	17118:
		F_ADSErrorCodeExt := 'Coupling conditions of synchronization generator incorrect';

	17119:
		F_ADSErrorCodeExt := 'Moving profile of synchronization generator declines dynamic limit of slave axis or required characteristic of profile';

	17120:
		F_ADSErrorCodeExt := 'The encoder generator parameter is not allowed.';

	17121:
		F_ADSErrorCodeExt := 'The external (Fifo) generator parameter is not allowed.';

	17122:
		F_ADSErrorCodeExt := 'The external generator cannot be started, as it is already active.';

	17123:
		F_ADSErrorCodeExt := 'The external generator cannot be stopped, as it is not active.';

	17124:
		F_ADSErrorCodeExt := 'NC-Block with auxiliary axis violates software limit switches of the group.';

	17125:
		F_ADSErrorCodeExt := 'NC-Block type Bezier spline curve contains a cusp (singularity). The Bezier spline curve contain a cusp.';

	17127:
		F_ADSErrorCodeExt := 'Value FOR dead TIME compensation NOT allowed.';

	17128:
		F_ADSErrorCodeExt := 'GROUPERR_RANGE_NOMOTIONWINDOW';

	17129:
		F_ADSErrorCodeExt := 'GROUPERR_RANGE_NOMOTIONFILTERTIME';

	17130:
		F_ADSErrorCodeExt := 'GROUPERR_RANGE_TIMEUNITFIFO';

	17131:
		F_ADSErrorCodeExt := 'GROUPERR_RANGE_OVERRIDETYPE';

	17132:
		F_ADSErrorCodeExt := 'GROUPERR_RANGE_OVERRIDECHANGETIME';

	17133:
		F_ADSErrorCodeExt := 'GROUPERR_FIFO_INVALIDDIMENSION';

	17134:
		F_ADSErrorCodeExt := 'GROUPERR_ADDR_FIFOTABLE';

	17135:
		F_ADSErrorCodeExt := 'Axis is locked for motion commands because a stop command is still active.';

	17136:
		F_ADSErrorCodeExt := 'Invalid number of auxiliary axes.';

	17137:
		F_ADSErrorCodeExt := 'The velocity reduction parameters FOR the auxiliary axes are inconsistent.';

	17138:
		F_ADSErrorCodeExt := 'The dynamic parameters FOR the auxiliary axes are inconsistent.';

	17139:
		F_ADSErrorCodeExt := 'The coupling parameters FOR the auxiliary axes are inconsistent.';

	17140:
		F_ADSErrorCodeExt := 'The auxiliary axis entry is empty (no axis motion).';

	17142:
		F_ADSErrorCodeExt := 'The LIMIT FOR velocity reduction OF the auxiliary axes is invalid.';

	17144:
		F_ADSErrorCodeExt := 'Block search - segment NOT found. The segment specified as a parameter could not be found by the end of the NC program.';

	17145:
		F_ADSErrorCodeExt := 'Blocksearch – invalid remaining segment length. The remaining travel in the parameter fLength is incorrectly parameterized.';

	17147:
		F_ADSErrorCodeExt := 'INTERNAL Error in the Context OF Coupled Axes (Slave Axes).';

	17148:
		F_ADSErrorCodeExt := 'Parameter FOR the Maximum Number OF Jobs (Entries) TO be Transferred is Invalid';

	17151:
		F_ADSErrorCodeExt := 'Customer Specific Error';

	// NC - Axis Error Codes (Includes TF5055 Flying Saw)

	// 17152 - 17312)
	17152:
		F_ADSErrorCodeExt := 'Axis ID not allowed.';

	17153:
		F_ADSErrorCodeExt := 'Axis type not allowed.';

	17158:
		F_ADSErrorCodeExt := 'Slow manual velocity not allowed.';

	17159:
		F_ADSErrorCodeExt := 'Fast manual velocity not allowed.';

	17160:
		F_ADSErrorCodeExt := 'High speed not allowed.';

	17161:
		F_ADSErrorCodeExt := 'Acceleration not allowed.';

	17162:
		F_ADSErrorCodeExt := 'Deceleration not allowed.';

	17163:
		F_ADSErrorCodeExt := 'Jerk not allowed.';

	17164:
		F_ADSErrorCodeExt := 'Delay time between position and velocity is not allowed (dead time compensation).';

	17165:
		F_ADSErrorCodeExt := 'Override type not allowed.';

	17166:
		F_ADSErrorCodeExt := 'NCI: Velo-Jump-Factor not allowed.';

	17167:
		F_ADSErrorCodeExt := 'NCI: Size of tolerance sphere for auxiliary axis invalid.';

	17168:
		F_ADSErrorCodeExt := 'NCI: Value for maximum deviation for auxiliary axis invalid.';

	17170:
		F_ADSErrorCodeExt := 'Referencing velocity in direction of cam not allowed.';

	17171:
		F_ADSErrorCodeExt := 'Referencing velocity in sync direction not allowed.';

	17172:
		F_ADSErrorCodeExt := 'Pulse width in positive direction not allowed';

	17173:
		F_ADSErrorCodeExt := 'Pulse width in negative direction not allowed';

	17174:
		F_ADSErrorCodeExt := 'The value for the pulse width in positive direction is not allowed (pulsed operation).';

	17175:
		F_ADSErrorCodeExt := 'The value for the pulse width in negative direction is not allowed (pulsed operation).';

	17176:
		F_ADSErrorCodeExt := 'The value for the creep distance in positive direction is not allowed.';

	17177:
		F_ADSErrorCodeExt := 'The value for the creep distance in negative direction is not allowed.';

	17178:
		F_ADSErrorCodeExt := 'The value for the braking distance in positive direction is not allowed.';

	17179:
		F_ADSErrorCodeExt := 'The value for the braking distance in negative direction is not allowed.';

	17180:
		F_ADSErrorCodeExt := 'The value for the braking time in positive direction is not allowed.';

	17181:
		F_ADSErrorCodeExt := 'The value for the braking time in negative direction is not allowed.';

	17182:
		F_ADSErrorCodeExt := 'The value for the switching time from high to low speed is not allowed.';

	17183:
		F_ADSErrorCodeExt := 'The value for the creep distance for an explicit stop is not allowed.';

	17184:
		F_ADSErrorCodeExt := 'The value for the motion monitoring time is not allowed.';

	17185:
		F_ADSErrorCodeExt := 'The value for the activation of the position window monitoring is not allowed.';

	17186:
		F_ADSErrorCodeExt := 'The value for the activation of target window monitoring is not allowed.';

	17187:
		F_ADSErrorCodeExt := 'The value for the activation of loop movement is not allowed.';

	17188:
		F_ADSErrorCodeExt := 'The value for the motion monitoring time is not allowed.';

	17189:
		F_ADSErrorCodeExt := 'The value for the target window is not allowed.';

	17190:
		F_ADSErrorCodeExt := 'The value for the position window is not allowed.';

	17191:
		F_ADSErrorCodeExt := 'The value for the position window monitoring time is not allowed.';

	17192:
		F_ADSErrorCodeExt := 'The value for the loop movement is not allowed.';

	17193:
		F_ADSErrorCodeExt := 'The value for the axis cycle time is not allowed.';

	17194:
		F_ADSErrorCodeExt := 'The value for the stepper motor operating mode is not allowed.';

	17195:
		F_ADSErrorCodeExt := 'The value for the displacement associated with one step of the stepper motor is not allowed (step scaling).';

	17196:
		F_ADSErrorCodeExt := 'The value for the minimum speed of the stepper motor speed profile is not allowed.';

	17197:
		F_ADSErrorCodeExt := 'The value for the number of steps per speed level of the setpoint generation is not allowed.';

	17198:
		F_ADSErrorCodeExt := 'The value containing the flags for the interpretation of position and velocity units is not allowed.';

	17199:
		F_ADSErrorCodeExt := 'The value for the maximum permitted velocity is not allowed.';

	17200:
		F_ADSErrorCodeExt := 'The value for the motion monitoring window is not allowed.';

	17201:
		F_ADSErrorCodeExt := 'The value for the activation of the PEH time monitoring is not allowed (PEH: positioning end and halt).';

	17202:
		F_ADSErrorCodeExt := 'The value for the PEH monitoring time (timeout) is not allowed (PEH: positioning end and halt). Default value: 5s';

	17203:
		F_ADSErrorCodeExt := 'Parameter "Brake Release Delay" is invalid';

	17204:
		F_ADSErrorCodeExt := 'Parameter "NC Data Persistence" is invalid';

	17205:
		F_ADSErrorCodeExt := 'Parameter for Error Reaction Mode is invalid';

	17206:
		F_ADSErrorCodeExt := 'Parameter for the Error Reaction Delay is invalid';

	17207:
		F_ADSErrorCodeExt := 'Parameter "Use actual values in deactivated state" is invalid';

	17208:
		F_ADSErrorCodeExt := 'Parameter "Allow Motion Commands for Slave Axes" is invalid';

	17209:
		F_ADSErrorCodeExt := 'Parameter "Allow Motion Commands for axis in external setpoint generation" is invalid';

	17210:
		F_ADSErrorCodeExt := 'Parameter "Fading Acceleration" is invalid';

	17211:
		F_ADSErrorCodeExt := 'The value for the signal type of the Fast Axis Stop is not allowed [0...5].';

	17216:
		F_ADSErrorCodeExt := 'Axis has not been initialized.';

	17217:
		F_ADSErrorCodeExt := 'Axis does not have a group, or the group address has not been initialized (group contains the setpoint generation).';

	17218:
		F_ADSErrorCodeExt := 'The axis does not have an encoder, or the encoder address has not been initialized.';

	17219:
		F_ADSErrorCodeExt := 'An axis does not have a controller, or the controller address has not been initialized.';

	17220:
		F_ADSErrorCodeExt := 'The axis does not have a drive, or the drive address has not been initialized.';

	17221:
		F_ADSErrorCodeExt := 'Axis does not have an axis interface from the PLC to the NC, or the axis interface address has not been initialized.';

	17222:
		F_ADSErrorCodeExt := 'Axis does not have an axis interface from the NC to the PLC, or the axis interface address has not been initialized.';

	17223:
		F_ADSErrorCodeExt := 'The size of the axis interface from the NC to the PLC (NC to PLC) is not allowed.';

	17224:
		F_ADSErrorCodeExt := 'The size of the axis interface from the PLC to the NC is not allowed.';

	17238:
		F_ADSErrorCodeExt := 'Controller enable for the axis is not present.';

	17239:
		F_ADSErrorCodeExt := 'Missing negative feed enable for negative motion direction.';

	17240:
		F_ADSErrorCodeExt := 'Missing positive feed enable for positive motion direction.';

	17241:
		F_ADSErrorCodeExt := 'Set velocity not allowed.';

	17242:
		F_ADSErrorCodeExt := 'Movement smaller than one encoder increment not allowed';

	17243:
		F_ADSErrorCodeExt := 'The set acceleration has exceeded the maximum permitted acceleration or deceleration parameters of the axis';

	17244:
		F_ADSErrorCodeExt := 'The PEH time monitoring time that follows positioning has elapsed, the target position window has not been reached.';

	17245:
		F_ADSErrorCodeExt := 'The actual position of the axis has not changed or has changed only slightly during the motion monitoring time.';

	17246:
		F_ADSErrorCodeExt := 'Looping distance less than breaking distance.';

	17247:
		F_ADSErrorCodeExt := 'Starting velocity not allowed.';

	17248:
		F_ADSErrorCodeExt := 'Final velocity not allowed.';

	17249:
		F_ADSErrorCodeExt := 'Time range exceeded (future). The calculated position lies too far in the future.';

	17250:
		F_ADSErrorCodeExt := 'Time range exceeded (past)" The calculated position lies too far in the past.';

	17251:
		F_ADSErrorCodeExt := 'The requested position cannot be determined.';

	17252:
		F_ADSErrorCodeExt := 'Position indeterminable (conflicting direction of travel)';

	17264:
		F_ADSErrorCodeExt := 'No slave coupling possible (velocity violation)';

	17265:
		F_ADSErrorCodeExt := 'No slave coupling possible (acceleration violation)';

	17266:
		F_ADSErrorCodeExt := 'The synchronization profile would violate the lower end position of the slave.';

	17267:
		F_ADSErrorCodeExt := 'The synchronization profile would violate the upper end position of the slave.';

	17268:
		F_ADSErrorCodeExt := 'The synchronization profile would violate the user limit position Options.PositionLimitMin.';

	17269:
		F_ADSErrorCodeExt := 'The synchronization profile would violate the user limit position Options.PositionLimitMax.';

	17270:
		F_ADSErrorCodeExt := 'The synchronization point lies under the starting point. As a result, the profile swings under both the start position and the synchronous position.';

	17271:
		F_ADSErrorCodeExt := 'The synchronization profile would swing back under the slave start position of the flying saw.';

	17272:
		F_ADSErrorCodeExt := 'The synchronization point lies under the starting point. The synchronization profile would swing beyond the slave start position of the flying saw.';

	17273:
		F_ADSErrorCodeExt := 'The synchronization profile would swing beyond the slave synchronous position of the flying saw.';

	17274:
		F_ADSErrorCodeExt := 'The maximum velocity of the synchronization profile is higher than the maximum velocity of the slave axis.';

	17275:
		F_ADSErrorCodeExt := 'The maximum velocity of the synchronization profile is higher than the maximum velocity of the slave axis.';

	17276:
		F_ADSErrorCodeExt := 'The maximum velocity of the synchronization profile would be higher than the synchronous velocity.';

	17277:
		F_ADSErrorCodeExt := 'The maximum velocity of the synchronization profile would be higher than the starting velocity and synchronous velocity.';

	17278:
		F_ADSErrorCodeExt := 'The maximum velocity of the synchronization profile would be higher than the synchronous velocity.';

	17279:
		F_ADSErrorCodeExt := 'The maximum velocity of the synchronization profile would be higher than the starting velocity and synchronous velocity.';

	17280:
		F_ADSErrorCodeExt := 'The minimum velocity of the synchronization profile lies below the synchronous velocity.';

	17281:
		F_ADSErrorCodeExt := 'The minimum velocity of the synchronization profile lies below the starting velocity.';

	17282:
		F_ADSErrorCodeExt := 'The minimum velocity of the synchronization profile lies below the synchronous velocity.';

	17283:
		F_ADSErrorCodeExt := 'The minimum velocity of the synchronization profile lies below the starting velocity.';

	17286:
		F_ADSErrorCodeExt := 'The velocity of the flying saw swings below zero; the motion is reversed.';

	17287:
		F_ADSErrorCodeExt := 'The velocity of the flying saw swings below zero; the motion is reversed.';

	17288:
		F_ADSErrorCodeExt := 'The maximum acceleration of the synchronization profile would be higher than the maximum acceleration of the slave axis.';

	17289:
		F_ADSErrorCodeExt := 'The maximum deceleration of the synchronization profile would be higher than the maximum deceleration of the slave axis.';

	17290:
		F_ADSErrorCodeExt := 'The maximum jerk of the synchronization profile would be higher than the maximum jerk of the slave axis.';

	17291:
		F_ADSErrorCodeExt := 'The maximum jerk of the synchronization profile would be higher than the maximum jerk of the slave axis.';

	17312:
		F_ADSErrorCodeExt := 'Axis consequential error. Consequential error resulting from another causative error related to another axis.';

	// NC - Encoder Error Codes 

	// 17408 - 17571
	17408:
		F_ADSErrorCodeExt := 'Encoder ID NOT allowed';

	17409:
		F_ADSErrorCodeExt := 'Encoder type not allowed';

	17410:
		F_ADSErrorCodeExt := 'The value for the encoder (operating) mode is not allowed.';

	17411:
		F_ADSErrorCodeExt := 'Encoder counting direction inverted?';

	17412:
		F_ADSErrorCodeExt := 'The flag for the referencing status is not allowed.';

	17413:
		F_ADSErrorCodeExt := 'The value for the number of encoder increments for each physical rotation of the encoder is not allowed.';

	17414:
		F_ADSErrorCodeExt := 'The value for the scaling factor is not allowed.';

	17415:
		F_ADSErrorCodeExt := 'The value for the position offset of the encoder is not allowed.';

	17416:
		F_ADSErrorCodeExt := 'The value for the encoders modulo factor is not allowed.';

	17417:
		F_ADSErrorCodeExt := 'The value for the actual position filter time is not allowed (P-T1 filter).';

	17418:
		F_ADSErrorCodeExt := 'The value for the actual velocity filter time is not allowed (P-T1 filter).';

	17419:
		F_ADSErrorCodeExt := 'The value for the actual acceleration filter time is not allowed (P-T1 filter).';

	17420:
		F_ADSErrorCodeExt := 'The value of the SAF cycle time for the calculation of actual values is not allowed (e.g. is less than or equal to zero).';

	17421:
		F_ADSErrorCodeExt := 'Configuration of the selected units is invalid” E.g. settings for modulo position, velocity per minute etc. lead to an error.';

	17422:
		F_ADSErrorCodeExt := 'The value for the activation of the actual position correction ("measuring system error correction") is not allowed.';

	17423:
		F_ADSErrorCodeExt := 'The value for the actual position correction filter time is not allowed (P-T1 filter).';

	17424:
		F_ADSErrorCodeExt := 'Search direction for referencing cam inverted.';

	17425:
		F_ADSErrorCodeExt := 'Search direction for sync pulse (zero pulse) inverted.';

	17426:
		F_ADSErrorCodeExt := 'The value of the reference position in a referencing procedure is not allowed.';

	17427:
		F_ADSErrorCodeExt := 'Clearance monitoring between activation of the hardware latch and appearance of the sync pulse.';

	17428:
		F_ADSErrorCodeExt := 'Minimum clearance between activation of the hardware latch and appearance of the sync pulse.';

	17429:
		F_ADSErrorCodeExt := 'The value of the activation or deactivation of the external sync pulse in a referencing procedure is not allowed.';

	17430:
		F_ADSErrorCodeExt := 'Scaling of the noise rate on simulation encoder is not allowed.';

	17431:
		F_ADSErrorCodeExt := 'The value for the tolerance window for the modulo-axis-start is invalid.';

	17432:
		F_ADSErrorCodeExt := 'The value for the encoder reference mode is not allowed, resp. is not supported for this encoder type.';

	17433:
		F_ADSErrorCodeExt := 'The value for the encoder evaluation direction (log. counter direction) is not allowed.';

	17434:
		F_ADSErrorCodeExt := 'The value for the encoder reference system is invalid.';

	17435:
		F_ADSErrorCodeExt := 'When starting the TC system the value for the encoder position initialization mode is invalid.';

	17436:
		F_ADSErrorCodeExt := 'Encoder sign interpretation (UNSIGNED- / SIGNED- data type) is invalid.';

	17437:
		F_ADSErrorCodeExt := 'The value for the encoder homing sensor source is not allowed.';

	17440:
		F_ADSErrorCodeExt := 'Software minimum end location monitoring not allowed.';

	17441:
		F_ADSErrorCodeExt := 'Software maximum end location monitoring not allowed.';

	17442:
		F_ADSErrorCodeExt := 'Actual value setting is outside the value range.';

	17443:
		F_ADSErrorCodeExt := 'Software end location minimum not allowed.';

	17444:
		F_ADSErrorCodeExt := 'Software end location maximum not allowed.';

	17445:
		F_ADSErrorCodeExt := 'The value for the filter mask of the encoder raw data in increments is invalid.';

	17446:
		F_ADSErrorCodeExt := 'Reference mask for the raw data of the encoder is invalid';

	17447:
		F_ADSErrorCodeExt := 'Parameter Dead Time Compensation Mode (Encoder) is Invalid';

	17448:
		F_ADSErrorCodeExt := 'Parameter “Control Bits of Dead Time Compensation” (Encoder) is Invalid';

	17449:
		F_ADSErrorCodeExt := 'Parameter “Time Related Shift of Dead Time Compensation Mode” (Encoder) is Invalid';

	17456:
		F_ADSErrorCodeExt := 'Hardware latch activation (encoder), hardware latch was implicitly initated by the referencing procedure.';

	17457:
		F_ADSErrorCodeExt := 'External hardware latch activation (encoder) via ADS has already been activated, but no valid latch value present';

	17458:
		F_ADSErrorCodeExt := 'External hardware latch activation (encoder), hardware still signals a valid latch value.';

	17459:
		F_ADSErrorCodeExt := 'External hardware latch activation (encoder), hardware still signalling that the external latch value is still valid.';

	17460:
		F_ADSErrorCodeExt := 'An encoder function has been activated that is currently not released for use, or which is not even implemented.';

	17461:
		F_ADSErrorCodeExt := 'An encoder function can not been activated because this functionality is already active.';

	17472:
		F_ADSErrorCodeExt := 'Encoder has not been initialized.';

	17473:
		F_ADSErrorCodeExt := 'The encoder does not have an axis, or the axis address has not been initialized.';

	17474:
		F_ADSErrorCodeExt := 'The drive does not have a valid I/O input address in the process image.';

	17475:
		F_ADSErrorCodeExt := 'The encoder does not have a valid I/O output address in the process image.';

	17488:
		F_ADSErrorCodeExt := 'The encoders incremental counter has underflowed.';

	17489:
		F_ADSErrorCodeExt := 'The encoders incremental counter has overflowed.';

	17504:
		F_ADSErrorCodeExt := 'Minimum Software Position Limit (Axis Start).';

	17505:
		F_ADSErrorCodeExt := 'Maximum Software Position Limit (Axis Start).';

	17506:
		F_ADSErrorCodeExt := 'Minimum Software Position Limit (Positioning Process).';

	17507:
		F_ADSErrorCodeExt := 'Maximum Software Position Limit (Positioning Process).';

	17508:
		F_ADSErrorCodeExt := 'Encoder hardware error.';

	17509:
		F_ADSErrorCodeExt := 'Position initialization error at system start.';

	17510:
		F_ADSErrorCodeExt := 'Invalid IO data for more than n subsequent NC cycles (encoder)';

	17511:
		F_ADSErrorCodeExt := 'Invalid Actual Position (Encoder)';

	17512:
		F_ADSErrorCodeExt := 'Invalid IO Input Data (Error Type 1)';

	17513:
		F_ADSErrorCodeExt := 'Invalid IO Input Data (Error Type 2)';

	17520:
		F_ADSErrorCodeExt := 'SSI transformation fault or not finished.';

	17570:
		F_ADSErrorCodeExt := 'ENCERR_ADDR_CONTROLLER';

	17571:
		F_ADSErrorCodeExt := 'ENCERR_INVALID_CONTROLLERTYPE';

	// NC - Controller Error Codes 

	// 17664 - 17828
	17664:
		F_ADSErrorCodeExt := 'Controller ID not allowed.';

	17665:
		F_ADSErrorCodeExt := 'Controller type not allowed.';

	17666:
		F_ADSErrorCodeExt := 'Controller operating mode not allowed.';

	17667:
		F_ADSErrorCodeExt := 'The value for the percentage weighting of the velocity pre-control is not allowed. The parameter is pre-set to 1.0 (100%) as standard.';

	17668:
		F_ADSErrorCodeExt := 'The value for the activation of the following error monitoring is not allowed.';

	17669:
		F_ADSErrorCodeExt := 'The value for the activation of the following error monitoring (velocity) is not allowed.';

	17670:
		F_ADSErrorCodeExt := 'The value for the following error window (maximum allowable following error) is not allowed.';

	17671:
		F_ADSErrorCodeExt := 'The value for the following error filter time (position) is not allowed.';

	17672:
		F_ADSErrorCodeExt := 'The value for the following error window (velocity) is not allowed.';

	17673:
		F_ADSErrorCodeExt := 'The value for the following error filter time (velocity) is not allowed.';

	17674:
		F_ADSErrorCodeExt := '“Controller Output Limitation” Improper';

	17680:
		F_ADSErrorCodeExt := 'Proportional gain Kv or Kp (controller) not allowed.';

	17681:
		F_ADSErrorCodeExt := 'Integral-action time Tn (controller) not allowed.';

	17682:
		F_ADSErrorCodeExt := 'Derivative action time Tv (controller) not allowed.';

	17683:
		F_ADSErrorCodeExt := 'Damping time Td (controller) not allowed.';

	17684:
		F_ADSErrorCodeExt := 'Activation of the automatic offset compensation not allowed.';

	17685:
		F_ADSErrorCodeExt := 'Additional proportional gain Kv or Kp (controller) not allowed.';

	17686:
		F_ADSErrorCodeExt := 'Reference velocity for additional proportional gain Kv or Kp (controller) not allowed.';

	17687:
		F_ADSErrorCodeExt := 'Proportional gain Pa (proportion) not allowed.';

	17688:
		F_ADSErrorCodeExt := 'Proportional gain Kv (velocity controller) not allowed.';

	17689:
		F_ADSErrorCodeExt := 'Reset time Tn (velocity controller) not allowed.';

	17690:
		F_ADSErrorCodeExt := 'Reserved';

	17691:
		F_ADSErrorCodeExt := 'Reserved';

	17692:
		F_ADSErrorCodeExt := 'Velocity Filter Time” Improper';

	17693:
		F_ADSErrorCodeExt := 'Dead zone not allowed.';

	17695:
		F_ADSErrorCodeExt := 'Proportionality Factor Kcp” Improper.';

	17696:
		F_ADSErrorCodeExt := 'Rate time Tv (velocity controller) not allowed.';

	17697:
		F_ADSErrorCodeExt := 'Damping time Td (velocity controller) not allowed.';

	17698:
		F_ADSErrorCodeExt := 'Limitation of the I Part” Improper.';

	17699:
		F_ADSErrorCodeExt := 'Limitation of the D Part” Improper.';

	17700:
		F_ADSErrorCodeExt := 'Parameter “Switching Off the I Part During Motion” is Improper.';

	17701:
		F_ADSErrorCodeExt := 'Parameter “Filter Time for P-T2 Filter” Improper.';

	17702:
		F_ADSErrorCodeExt := 'Velocity Observer: “Parameterized Mode” is Improper.';

	17703:
		F_ADSErrorCodeExt := 'Velocity Observer: “Motor Torque Constant Kt or Kf” is Improper.';

	17704:
		F_ADSErrorCodeExt := 'Velocity Observer: “Motor Moment of Inertia JM” is Improper.';

	17705:
		F_ADSErrorCodeExt := 'Velocity Observer: “Band Width f0” is Improper.';

	17706:
		F_ADSErrorCodeExt := 'Velocity Observer: “Correction Factor kc” is Improper.';

	17707:
		F_ADSErrorCodeExt := 'Velocity Observer: “Time Constant T for First Order Filter” is Improper.';

	17708:
		F_ADSErrorCodeExt := 'Velocity Observer: “Amplitude Damping d for Second Order Filter” is Improper.';

	17709:
		F_ADSErrorCodeExt := 'Velocity Observer: “Frequency fHP or Frequency fTP for Filters of Second Order” is Improper.';

	17728:
		F_ADSErrorCodeExt := 'Controller has not been initialized.';

	17729:
		F_ADSErrorCodeExt := 'Controller does not know its axis, or the axis address has not been initialized.';

	17730:
		F_ADSErrorCodeExt := 'Controller does not know its drive, or the drive address has not been initialized.';

	17744:
		F_ADSErrorCodeExt := 'Following error monitoring (position). A following error exceedance has occurred';

	17745:
		F_ADSErrorCodeExt := 'Following error monitoring (velocity). A velocity following error exceedance has occurred';

	17824:
		F_ADSErrorCodeExt := 'CONTROLERR_RANGE_AREA_ASIDE';

	17825:
		F_ADSErrorCodeExt := 'CONTROLERR_RANGE_AREA_BSIDE';

	17826:
		F_ADSErrorCodeExt := 'CONTROLERR_RANGE_QNENN';

	17827:
		F_ADSErrorCodeExt := 'CONTROLERR_RANGE_PNENN';

	17828:
		F_ADSErrorCodeExt := 'CONTROLERR_RANGE_AXISIDPRESP0';

	// NC - Drive Error Codes 

	// 17920 - 18005
	17920:
		F_ADSErrorCodeExt := 'Drive ID not allowed.';

	17921:
		F_ADSErrorCodeExt := 'Drive type not allowed.';

	17922:
		F_ADSErrorCodeExt := 'Drive operation mode not allowed.';

	17923:
		F_ADSErrorCodeExt := 'Motor polarity inverted?.';

	17924:
		F_ADSErrorCodeExt := 'The value for the drift compensation (DAC offset) is not allowed.';

	17925:
		F_ADSErrorCodeExt := 'The value for the reference velocity (also called velocity pre-control) is not allowed.';

	17926:
		F_ADSErrorCodeExt := 'The value for the reference output in percent is not allowed. The value 1.0 (100 %) usually corresponds to a voltage of 10.0 V.';

	17927:
		F_ADSErrorCodeExt := 'The value for the quadrant compensation factor is not allowed.';

	17928:
		F_ADSErrorCodeExt := 'The value for the velocity reference point in percent is not allowed. The value 1.0 corresponds to 100 percent.';

	17929:
		F_ADSErrorCodeExt := 'The value for the output reference point in percent is not allowed. The value 1.0 corresponds to 100 percent.';

	17930:
		F_ADSErrorCodeExt := 'The value for the minimum and/or maximum drive output limit is not allowed.';

	17931:
		F_ADSErrorCodeExt := 'Parameter "Maximum value for output" is not allowed';

	17932:
		F_ADSErrorCodeExt := 'Parameter "Internal Drive Control Word" is not allowed';

	17933:
		F_ADSErrorCodeExt := 'Parameter "Internal timer for RESET behavior Drive" is not allowed';

	17934:
		F_ADSErrorCodeExt := 'Parameter "Master Motion Controller ID" is not allowed';

	17935:
		F_ADSErrorCodeExt := 'Drive torque output scaling not allowed.';

	17936:
		F_ADSErrorCodeExt := 'Drive velocity output scaling not allowed.';

	17937:
		F_ADSErrorCodeExt := 'Profi Drive DSC proportional gain Kpc (controller) not allowed.';

	17938:
		F_ADSErrorCodeExt := 'The value for the table ID is not allowed.';

	17939:
		F_ADSErrorCodeExt := 'The value is not allowed as the table interpolation type.';

	17940:
		F_ADSErrorCodeExt := 'The value is not allowed as an output offset in percent (+/- 1.0).';

	17941:
		F_ADSErrorCodeExt := 'Profi Drive DSC scaling for calculation of "Xerr" (controller) not allowed.';

	17942:
		F_ADSErrorCodeExt := 'The value is not allowed as drive acceleration/deceleration output scaling.';

	17943:
		F_ADSErrorCodeExt := 'The value is not allowed as drive position output scaling.';

	17944:
		F_ADSErrorCodeExt := 'Parameter "Dead time compensation mode" (Motion Controller) is invalid';

	17945:
		F_ADSErrorCodeExt := 'Parameter "Control bits of the dead time compensation" (Motion Controller) is invalid';

	17946:
		F_ADSErrorCodeExt := 'Parameter "time shift of dead time compensation mode" (Motion Controller) is invalid';

	17947:
		F_ADSErrorCodeExt := 'Parameter "Output delay velocity interface Motion Controller" is invalid';

	17948:
		F_ADSErrorCodeExt := 'Drive filter type not allowed for command variable filter for the output position.';

	17949:
		F_ADSErrorCodeExt := 'Drive filter time not allowed for command variable filter for the output position.';

	17950:
		F_ADSErrorCodeExt := 'The value is not allowed as a drive filter order (P-Tn) for the smoothing of the output position (command variable filter for the set position).';

	17952:
		F_ADSErrorCodeExt := 'Bit mask for stepper motor cycle not allowed.';

	17953:
		F_ADSErrorCodeExt := 'Bit mask for stepper motor holding current not allowed.';

	17954:
		F_ADSErrorCodeExt := 'Scaling factor for actual torque (actual current) not allowed.';

	17955:
		F_ADSErrorCodeExt := 'Filter time for actual torque is not allowed.';

	17956:
		F_ADSErrorCodeExt := 'Filter time for the temporal derivation of the actual torque is not allowed.';

	17957:
		F_ADSErrorCodeExt := 'Parameter "Drive operation mode" is invalid';

	17958:
		F_ADSErrorCodeExt := 'Motion Controller function is not supported';

	17959:
		F_ADSErrorCodeExt := 'The activation of the drive operation mode failed, because another object with OID… is already using this interface.';

	17960:
		F_ADSErrorCodeExt := 'Drive operation mode changeover is not configured or the desired drive operation mode cannot be found';

	17961:
		F_ADSErrorCodeExt := 'Feedback drive operation mode changeover';

	17968:
		F_ADSErrorCodeExt := 'Overtemperature" Overtemperature was detected or reported in the drive or terminal.';

	17969:
		F_ADSErrorCodeExt := 'Undervoltage was detected or reported in the drive or terminal.';

	17970:
		F_ADSErrorCodeExt := 'Open circuit in phase A.';

	17971:
		F_ADSErrorCodeExt := 'Open circuit in phase B.';

	17972:
		F_ADSErrorCodeExt := 'Overcurrent in phase A.';

	17973:
		F_ADSErrorCodeExt := 'Overcurrent in phase B.';

	17974:
		F_ADSErrorCodeExt := 'A torque overload (stall) was detected or reported in the drive or terminal.';

	17984:
		F_ADSErrorCodeExt := 'Drive has not been initialized.';

	17985:
		F_ADSErrorCodeExt := 'Drive does not know its axis, or the axis address has not been initialized.';

	17986:
		F_ADSErrorCodeExt := 'Drive has no valid I/O input address in the process image.';

	17987:
		F_ADSErrorCodeExt := 'Drive has no valid I/O output address in the process image.';

	18000:
		F_ADSErrorCodeExt := 'The drive hardware is not ready for operation.';

	18001:
		F_ADSErrorCodeExt := 'Error in the cyclic communication of the drive (Life Counter). Reasons for this could be an interrupted fieldbus or a drive that is in the error state.';

	18002:
		F_ADSErrorCodeExt := 'Changing the table ID when active controller enable is not allowed.';

	18005:
		F_ADSErrorCodeExt := 'Invalid I/O data for more than "n" continuous NC cycles.';

	// NC - Table Error Codes

	// 18944 - 18981
	18944:
		F_ADSErrorCodeExt := 'Table ID not allowed.';

	18945:
		F_ADSErrorCodeExt := 'Table type not allowed.';

	18946:
		F_ADSErrorCodeExt := 'Number of lines in the table not allowed.';

	18947:
		F_ADSErrorCodeExt := 'Number of columns in the table is not allowed.';

	18948:
		F_ADSErrorCodeExt := 'Step size (position delta) not allowed.';

	18949:
		F_ADSErrorCodeExt := 'Period not allowed.';

	18950:
		F_ADSErrorCodeExt := 'Table is not monotonic.';

	18951:
		F_ADSErrorCodeExt := 'Table sub type is not allowed.';

	18952:
		F_ADSErrorCodeExt := 'Table interpolation type is not allowed.';

	18953:
		F_ADSErrorCodeExt := 'The table main type is unknown or otherwise the table class (slave type) do not match up to the table main type.';

	18960:
		F_ADSErrorCodeExt := 'Table has not been initialized.';

	18961:
		F_ADSErrorCodeExt := 'Table could not be created, since there is not enough memory.';

	18962:
		F_ADSErrorCodeExt := 'The function has not been implemented, or cannot be executed, for the present type of table.';

	18963:
		F_ADSErrorCodeExt := 'The start line index or the stop line index to be used for read or write access to the table is not allowed.';

	18964:
		F_ADSErrorCodeExt := 'The start column index or the stop column index to be used for read or write access to the table in not allowed.';

	18965:
		F_ADSErrorCodeExt := 'The number of lines to be read from or written to the table is not allowed.';

	18966:
		F_ADSErrorCodeExt := 'The number of columns to be read from or written to the table is not allowed.';

	18967:
		F_ADSErrorCodeExt := 'The entries in the table header are inconsistent, e.g. the validity range is empty.';

	18968:
		F_ADSErrorCodeExt := 'The slave master position is outside the table values for the master.';

	18969:
		F_ADSErrorCodeExt := 'Solo table underflow. The slave master position is outside the table values for the master.';

	18970:
		F_ADSErrorCodeExt := 'Solo table overflow. The slave master position is outside the table values for the master.';

	18971:
		F_ADSErrorCodeExt := 'Incorrect execution mode.';

	18972:
		F_ADSErrorCodeExt := 'Impermissible parameter. The Fifo parameter is not allowed.';

	18973:
		F_ADSErrorCodeExt := 'Fifo is empty.';

	18974:
		F_ADSErrorCodeExt := 'Fifo is full.';

	18975:
		F_ADSErrorCodeExt := 'Point-Index of Motion Function invalid.';

	18976:
		F_ADSErrorCodeExt := 'No diagonalisation of  matrix. The spline can not be calculated.';

	18977:
		F_ADSErrorCodeExt := 'The number of points of a cubic spline has to be greater than two.';

	18978:
		F_ADSErrorCodeExt := 'Fifo must not be overwritten.';

	18979:
		F_ADSErrorCodeExt := 'Insufficient number of Motion Function points.';

	18981:
		F_ADSErrorCodeExt := 'A periodic position table must start with a master position zero.';

	// NC - NC-PLC Error Codes

	// 19200 - 19395
	19200:
		F_ADSErrorCodeExt := 'The axis was stopped during travel to the target position.';

	19201:
		F_ADSErrorCodeExt := 'Axis cannot be started. Error, or busy, or protected, or not ready for operation.';

	19202:
		F_ADSErrorCodeExt := 'No target position control, and no position range control permitted.';

	19203:
		F_ADSErrorCodeExt := 'The position and velocity can only be restarted while the axis is physically in motion.';

	19204:
		F_ADSErrorCodeExt := 'Invalid mode. Invalide Direction with MC_MoveModulo, or inactive axis parameter "Position Correction" with MC_BacklashCompensation.';

	19205:
		F_ADSErrorCodeExt := 'Command not permitted. Direction not specified, or read/write parameter type mismatch.';

	19206:
		F_ADSErrorCodeExt := 'Parameter incorrect. Override outside bounds, or read/write parameter type mismatch.';

	19207:
		F_ADSErrorCodeExt := 'Timeout axis function block. Position range monitoring time exceeded, target position monitoring time exceeded.';

	19208:
		F_ADSErrorCodeExt := 'The axis is in protected mode (e.g., coupled) and cannot be moved.';

	19209:
		F_ADSErrorCodeExt := 'Axis is not ready.';

	19210:
		F_ADSErrorCodeExt := 'Error during referencing.';

	19211:
		F_ADSErrorCodeExt := 'The definition of the trigger signal for function block MC_TouchProbe is incorrect..';

	19212:
		F_ADSErrorCodeExt := 'Position latch was disabled after MC_Touchprobe execute.';

	19213:
		F_ADSErrorCodeExt := 'NC status feedback timeout. An expected feedback in the axis status word has not arrived.';

	19214:
		F_ADSErrorCodeExt := 'Additional product not installed.';

	19215:
		F_ADSErrorCodeExt := 'No NC Cycle Counter Update.';

	19216:
		F_ADSErrorCodeExt := 'M-function query missing.';

	19217:
		F_ADSErrorCodeExt := 'Zero shift index is outside the range. The index of the zero shift is invalid.';

	19218:
		F_ADSErrorCodeExt := 'R-parameter index or size is invalid. This error occurs if the R-parameters are written or read but the index or size are outside the range.';

	19219:
		F_ADSErrorCodeExt := 'Index for tool description is invalid.';

	19220:
		F_ADSErrorCodeExt := 'Version of the cyclic channel interface does not match the requested function or the function block.';

	19221:
		F_ADSErrorCodeExt := 'Channel is not ready for the requested function.';

	19222:
		F_ADSErrorCodeExt := 'The requested function requires explicit activation.';

	19223:
		F_ADSErrorCodeExt := 'Axis is already in another group.';

	19224:
		F_ADSErrorCodeExt := 'Block search could not be executed successfully.';

	19225:
		F_ADSErrorCodeExt := 'This error occurs if the FB ItpBlocksearch is called with invalid parameters (e.g., E_ItpDryRunMode, E_ItpBlockSearchMode)';

	19232:
		F_ADSErrorCodeExt := 'Cannot add all axes to the interpolation group.';

	19248:
		F_ADSErrorCodeExt := 'A pointer to a data structure is invalid, e.g., Null';

	19249:
		F_ADSErrorCodeExt := 'The specification of the memory size (SIZE) for a data structure is invalid.';

	19250:
		F_ADSErrorCodeExt := 'Cam table ID is invalid.';

	19251:
		F_ADSErrorCodeExt := 'Point ID is invalid. The ID of a point (sampling point) of a motion function is less than 1.';

	19252:
		F_ADSErrorCodeExt := 'The number of points (sampling points) of a cam plate to be read or written is less than 1.';

	19253:
		F_ADSErrorCodeExt := 'The type of a cam plate does not match the definition MC_TableType.';

	19254:
		F_ADSErrorCodeExt := 'The number of rows (sampling points) of a cam table is less than 1.';

	19255:
		F_ADSErrorCodeExt := 'The number of columns of a cam table is invalid.';

	19256:
		F_ADSErrorCodeExt := 'Step size invalid. The increment for the interpolation is invalid, e.g., less than or equal to zero.';

	19264:
		F_ADSErrorCodeExt := 'The terminal used is not supported by this function block.';

	19265:
		F_ADSErrorCodeExt := 'Register read/write error. This error implies a validity error.';

	19266:
		F_ADSErrorCodeExt := 'The axis is enabled but should not be enabled for this process.';

	19267:
		F_ADSErrorCodeExt := 'Incorrect size of the compensation table. The specified table size (in bytes) does not match the actual size';

	19268:
		F_ADSErrorCodeExt := 'The minimum/maximum position in the compensation table does not match the position in the table description (ST_CompensationDesc)';

	19269:
		F_ADSErrorCodeExt := 'The requested function is not implemented in this combination';

	19270:
		F_ADSErrorCodeExt := 'Window not in the specified modulo range.';

	19271:
		F_ADSErrorCodeExt := 'Buffer overflow. The number of events has led to an overflow of the buffer and not all events could be acquired.';

	19296:
		F_ADSErrorCodeExt := 'Motion command did not become active.';

	19297:
		F_ADSErrorCodeExt := 'Motion command could not be monitored by the PLC.';

	19298:
		F_ADSErrorCodeExt := 'A buffered command was terminated with an error.';

	19299:
		F_ADSErrorCodeExt := 'A buffered command was completed but there was no feedback to indicate success or failure.';

	19300:
		F_ADSErrorCodeExt := 'The BufferMode is not supported by this command.';

	19301:
		F_ADSErrorCodeExt := 'The command number for queued commands managed by the system unexpectedly has the value 0.';

	19302:
		F_ADSErrorCodeExt := 'Function block was not called cyclically.';

	19313:
		F_ADSErrorCodeExt := 'Invalid NCI entry type. The FB FB_NciFeedTablePreparation was called with an unknown nEntryType.';

	19314:
		F_ADSErrorCodeExt := 'NCI feed table is full and the entry is therefore not accepted.';

	19315:
		F_ADSErrorCodeExt := 'Internal error.';

	19316:
		F_ADSErrorCodeExt := 'ST_NciTangentialFollowingDesc: Tangential axis is not an auxiliary axis.';

	19317:
		F_ADSErrorCodeExt := 'ST_NciTangentialFollowingDesc: nPathAxis1 or nPathAxis2 is not a path axis. It is therefore not possible to determine the plane.';

	19318:
		F_ADSErrorCodeExt := 'ST_NciTangentialFollwoingDesc: nPathAxis1 and nPathAxis2 are the same. It is therefore not possible to determine the plane.';

	19319:
		F_ADSErrorCodeExt := 'ST_NciGeoCirclePlane: Circle incorrectly parameterized';

	19320:
		F_ADSErrorCodeExt := 'Internal error during calculation of tangential following';

	19321:
		F_ADSErrorCodeExt := 'Tangential following: Monitoring of the deviation angle was activated during activation of tangential following.';

	19322:
		F_ADSErrorCodeExt := 'Not implemented';

	19323:
		F_ADSErrorCodeExt := 'Tangential following: the radius of the current arc is too small';

	19324:
		F_ADSErrorCodeExt := 'FB_NciFeedTablePreparation: pEntry is NULL';

	19325:
		F_ADSErrorCodeExt := 'FB_NciFeedTablePreparation: the specified nEntryType does not match the structure type';

	19326:
		F_ADSErrorCodeExt := 'ST_NciMFuncFast and ST_NciMFuncHsk: the requested M-function is not between 0 and 159';

	19327:
		F_ADSErrorCodeExt := 'ST_NciDynOvr: the requested value for the dynamic override is not between 0.01 and 1';

	19328:
		F_ADSErrorCodeExt := 'ST_NciVertexSmoothing: invalid parameter. This error is generated if a negative smoothing radius or an unknown smoothing type is encountered.';

	19329:
		F_ADSErrorCodeExt := 'FB_NciFeedTablePrepartion: The requested velocity is not in the valid range';

	19330:
		F_ADSErrorCodeExt := 'ST_Nci*: invalid parameter';

	19344:
		F_ADSErrorCodeExt := 'Determined drive type is not supported';

	19345:
		F_ADSErrorCodeExt := 'Direction is impermissible';

	19346:
		F_ADSErrorCodeExt := 'SwitchMode is impermissible';

	19347:
		F_ADSErrorCodeExt := 'Mode for the parameter handling is impermissible';

	19348:
		F_ADSErrorCodeExt := 'Parameterization of the torque limits is inconsistent';

	19349:
		F_ADSErrorCodeExt := 'Parameterization of the position lag limit is impermissible (<=0).';

	19350:
		F_ADSErrorCodeExt := 'Parameterization of the distance limit is impermissible (<0)';

	19351:
		F_ADSErrorCodeExt := 'An attempt was made to back up parameters again, although they have already been backed up.';

	19352:
		F_ADSErrorCodeExt := 'An attempt was made to restore parameters, although none have been backed up.';

	19359:
		F_ADSErrorCodeExt := 'The abortion of a homing has failed.';

	19360:
		F_ADSErrorCodeExt := 'KinGroup error: the kinematic group is in an error state.';

	19361:
		F_ADSErrorCodeExt := 'KinGroup timeout: timeout during call of a kinematic block';

	19376:
		F_ADSErrorCodeExt := 'The current axis position or the axis position resulting from the new position offset exceeds the valid range of values.';

	19377:
		F_ADSErrorCodeExt := 'The new position offset exceeds the valid range of values [AX5000: 2^31].';

	19378:
		F_ADSErrorCodeExt := 'The current axis position or the axis position resulting from the new position offset falls below the valid range of values.';

	19379:
		F_ADSErrorCodeExt := 'The new position offset falls below the valid range of values [AX5000: -2^31].';

	19380:
		F_ADSErrorCodeExt := 'The activated feedback and/or storage location (AX5000: P-0-0275) differ from the parameterization on the function block.';

	19381:
		F_ADSErrorCodeExt := 'Reinitialization of the actual NC position has failed, e.g., reference system = “ABSOLUTE (with single overflow)” & software end position monitoring is disabled.';

	19382:
		F_ADSErrorCodeExt := 'The command to set or delete a position offset was rejected without feedback data, e.g., if the drive controllers firmware does not support the corresponding command.';

	19383:
		F_ADSErrorCodeExt := 'The command to set or delete a position offset was rejected with feedback data. The information in the feedback data may contain further information about the cause.';

	19384:
		F_ADSErrorCodeExt := 'A firmware version >= 19 is required for the servo terminal.';

	19385:
		F_ADSErrorCodeExt := 'The modulo settings on the drive controller and NC are different.';

	19394:
		F_ADSErrorCodeExt := 'The new position offset exceeds the valid value range.';

	19395:
		F_ADSErrorCodeExt := 'I/O data are invalid or the terminal is in an error state.';

	// TF6310 TCP/IP

	// 32769 - 32773
	32769:
		F_ADSErrorCodeExt := 'No new sockets can be created (for FB_SocketListen and FB_SocketConnect)';

	32770:
		F_ADSErrorCodeExt := 'Socket handle is invalid (for FB_SocketReceive, FB_SocketAccept, FB_SocketSend etc.)';

	32771:
		F_ADSErrorCodeExt := 'TcpIp port listener already exists (returned from FB_SocketListen)';

	32772:
		F_ADSErrorCodeExt := 'Client socket is no longer connected with the server (returned from FB_SocketReceive)';

	32773:
		F_ADSErrorCodeExt := 'Error was registered in the listener socket (returned from FB_SocketAccept)';

	// Win32 Errors	
	16#8007274C:
		F_ADSErrorCodeExt := CONCAT('Win32 system error - ', 'A connection attempt failed because the connected party did not properly respond after a period of time, or the established connection failed because the connected host failed to respond.');

ELSE
	IF ErrorId >= 16#80070000 AND ErrorId <= 16#8007FFFF THEN
		CONCAT(CONCAT('Win32 system error - ', TO_STRING(ErrorId)), ', Not Found');
	ELSE
		IF ErrorId = 33056 THEN
			F_ADSErrorCodeExt := 'Invalid configuration for Object (e.g. in System Manager).';
		ELSIF ErrorId = 33057 THEN
			F_ADSErrorCodeExt := 'Invalid environment for Object (e.g. TcCom-Objects Hierarchy or missing/faulty Objects).';
		elsif ErrorId = 33058 Then
			F_ADSErrorCodeExt := 'Incompatible Driver or Object.';
		elsif ErrorId = 33060 Then
			F_ADSErrorCodeExt := 'Command execution does not terminate (e. g. MC_Reset does not signal DONE).';
		elsif ErrorId = 33072 Then
			F_ADSErrorCodeExt := 'Invalid ObjectID of Communication Target.';
		elsif ErrorId = 33073 Then
			F_ADSErrorCodeExt := 'Communication Target expects Call in different Context.';
		elsif ErrorId = 33074 Then
			F_ADSErrorCodeExt := 'Invalid State of Communication Target.';
		elsif ErrorId = 33076 Then
			F_ADSErrorCodeExt := 'Communication with Communication Target cannot be established.';
		elsif ErrorId = 33083 Then
			F_ADSErrorCodeExt := 'Transition Mode is invalid.';
		elsif ErrorId = 33084 Then
			F_ADSErrorCodeExt := 'BufferMode is invalid.';
		elsif ErrorId = 33085 Then
			F_ADSErrorCodeExt := 'Only one active Instance of Function Block per Group is allowed.';
		elsif ErrorId = 33086 Then
			F_ADSErrorCodeExt := 'Command is not allowed in current group state.';
		elsif ErrorId = 33087 Then
			F_ADSErrorCodeExt := 'Slave cannot synchronize. The slave cannot reach the SlaveSyncPosition with the given dynamics.';
		elsif ErrorId = 33088 Then
			F_ADSErrorCodeExt := 'Invalid value for one or more of the dynamic parameters (Acceleration, Deceleration, Jerk).';
		elsif ErrorId = 33089 Then
			F_ADSErrorCodeExt := 'IdentInGroup is invalid.';
		elsif ErrorId = 33090 Then
			F_ADSErrorCodeExt := 'The number of axes in the group is incompatible with the axes convention.';
		elsif ErrorId = 33091 Then
			F_ADSErrorCodeExt := 'Function Block or respective Command is not supported by Target.';
		elsif ErrorId = 33092 Then
			F_ADSErrorCodeExt := 'Command queue full. Command queue is completely filled up and cannot accept additional commands until some commands are fully processed.';
		elsif ErrorId = 33093 Then
			F_ADSErrorCodeExt := 'Mapping of Cyclic Interface between NC and PLC is missing (e.g. AXIS_REF, AXES_GROUP_REF, ...).';
		elsif ErrorId = 33094 Then
			F_ADSErrorCodeExt := 'Invalid Velocity Value. The velocity was not set or the entered value is invalid.';
		elsif ErrorId = 33095 Then
			F_ADSErrorCodeExt := 'Invalid Coordinate Dimension. The dimension of the set coordinate interpretation does not meet the requirements.';
		elsif ErrorId = 33096 Then
			F_ADSErrorCodeExt := 'Invalid Input Value.';
		elsif ErrorId = 33097 Then
			F_ADSErrorCodeExt := 'Unsupported Dynamics for selected Group Kernel.';
		elsif ErrorId = 33098 Then
			F_ADSErrorCodeExt := 'The programmed position dimension incompatible with the axes convention.';
		elsif ErrorId = 33099 Then
			F_ADSErrorCodeExt := 'Path buffer is invalid. E.g. because provided buffer has invalid address or is not big enough.';
		elsif ErrorId = 33100 Then
			F_ADSErrorCodeExt := 'Path does not contain any element.';
		elsif ErrorId = 33101 Then
			F_ADSErrorCodeExt := 'Provided Path buffer is too small to store more Path Elements.';
		elsif ErrorId = 33102 Then
			F_ADSErrorCodeExt := 'Dimension or at least one Value of Transition Parameters is invalid.';
		elsif ErrorId = 33103 Then
			F_ADSErrorCodeExt := 'Invalid or Incomplete Input Array.';
		elsif ErrorId = 33104 Then
			F_ADSErrorCodeExt := 'Path length is zero.';
		elsif ErrorId = 33105 Then
			F_ADSErrorCodeExt := 'Command is not allowed in current axis state.';
		elsif ErrorId = 33106 Then
			F_ADSErrorCodeExt := 'TwinCAT System is shutting down and cannot complete request.';
		elsif ErrorId = 33107 Then
			F_ADSErrorCodeExt := 'Configured axes convention and configured axes do not match.';
		elsif ErrorId = 33108 Then
			F_ADSErrorCodeExt := 'Invalid Number of ACS Axes. The number of ACS input axes does not match the number of ACS input axes expected by the kinematic transformation.';
		elsif ErrorId = 33109 Then
			F_ADSErrorCodeExt := 'Invalid Number of MCS Data. The number of MCS input data does not match the number expected by the kinematic transformation.';
		elsif ErrorId = 33110 Then
			F_ADSErrorCodeExt := 'Invalid Value Set for Kinematic Parameters. The numeric value set for the parameter does not reside within the respective definition range.';
		elsif ErrorId = 33112 Then
			F_ADSErrorCodeExt := 'The Given ACS Values Cannot be Reached. The given ACS values result in an invalid machine configuration.';
		elsif ErrorId = 33113 Then
			F_ADSErrorCodeExt := 'The Set Target Positions Cannot be Reached. The set target positions reside outside the admissible working space.';
		elsif ErrorId = 33117 Then
			F_ADSErrorCodeExt := 'Discontinuity in ACS axes detected.';
		elsif ErrorId = 33120 Then
			F_ADSErrorCodeExt := 'Circle Specification in Path is invalid. The specification of a circle segment in the programmed interpolated path (e.g. via MC_MovePath) has an invalid or ambiguous description. Probably its center cannot be determined reliably.';
		elsif ErrorId = 33121 Then
			F_ADSErrorCodeExt := 'Maximum stream lines reached. The maximum number of stream lines is limited. Please refer to function block documentation for details.';
		elsif ErrorId = 33123 Then
			F_ADSErrorCodeExt := 'Invalid First Segment. The corresponding element can only be analyzed with a well-defined start point.';
		elsif ErrorId = 33124 Then
			F_ADSErrorCodeExt := 'Invalid auxiliary point. The auxiliary point is not well-defined.';
		elsif ErrorId = 33126 Then
			F_ADSErrorCodeExt := 'Invalid parameter for GapControlMode. Invalid parameter for GapControlMode, most likely in combination with the group parameter GapControlDirection.';
		elsif ErrorId = 33127 Then
			F_ADSErrorCodeExt := 'Group got unsupported Axis Event (e.g. State Change). Group got unsupported Axis Event (e.g. State Change e.g. triggered by a Single Axis Reset).';
		elsif ErrorId = 33128 Then
			F_ADSErrorCodeExt := 'Unsupported Compensation Type. The compensation type was either not set or is not supported by the addressed object.';
		elsif ErrorId = 33129 Then
			F_ADSErrorCodeExt := 'Master axis does not exist or cannot be used.';
		elsif ErrorId = 33130 Then
			F_ADSErrorCodeExt := 'Invalid or Missing Tracking Transformation. This error occurs at MC_TrackConveyorBelt if at the CoordTransform input an invalid object ID is used or the object ID points to an object that is not supported as coordinate transformation.';
		elsif ErrorId = 33131 Then
			F_ADSErrorCodeExt := 'Position is not on Track. Either Track cannot be activated because Actual Position is not on Track, or Target Position is not on Active Track or TrackPart.';
		elsif ErrorId = 33132 Then
			F_ADSErrorCodeExt := 'Axis does not have an activated track.';
		elsif ErrorId = 33133 Then
			F_ADSErrorCodeExt := 'Invalid Compensation ObjectId. An Object with this ObjectId does not exist or it is not of the right type (has to be a compensation).';
		elsif ErrorId = 33134 Then
			F_ADSErrorCodeExt := 'Axis is in error because axis was not in Target when InTargetAlarm Timer expired.';
		elsif ErrorId = 33135 Then
			F_ADSErrorCodeExt := 'Coupling would cause a cyclic dependency of axis (e.g. via MC_GearInPos).';
		elsif ErrorId = 33136 Then
			F_ADSErrorCodeExt := 'Axis was not added to an axes group, the command is not valid.';
		elsif ErrorId = 33151 Then
			F_ADSErrorCodeExt := 'Drive has invalid State.';
		elsif ErrorId = 33153 Then
			F_ADSErrorCodeExt := 'Parameter for gap control are invalid with the current configuration. Function block with gap control was issued to an axis that is not in a CA group.';
		elsif ErrorId = 33154 Then
			F_ADSErrorCodeExt := 'Software position limit violation. Software position limits of at least one axis have been or would have been violated by a command.';
		elsif ErrorId = 33155 Then
			F_ADSErrorCodeExt := 'Target position is not reachable. There is no path available to the target position or target position is unreachable in general.';
		elsif ErrorId = 33157 Then
			F_ADSErrorCodeExt := 'The mover or one of its relevant coordinates is busy. Either the whole mover or at least of its coordinates relevant to the command are busy.';
		elsif ErrorId = 33158 Then
			F_ADSErrorCodeExt := 'A collision has occurred or would occur. Either a collision has occurred or would occur if the command was executed.';
		elsif ErrorId = 33159 Then
			F_ADSErrorCodeExt := 'Invalid Track Specification. The geometric extension of this track is incompatible with the already existing geometry of this or the other tracks.';
		elsif ErrorId = 33160 Then
			F_ADSErrorCodeExt := 'Command not allowed in track state.';
		elsif ErrorId = 33161 Then
			F_ADSErrorCodeExt :=
				'Invalid Reference passed to Function Block. An invalid reference (or pointer) was used in a function block call. This can happen if a reference type is used before it was initialized.';
		elsif ErrorId = 33162 Then
			F_ADSErrorCodeExt := 'Path is locked against modifications. The path was locked to further changes. However, it might be resettable.';
		ELSIF ErrorId = 33164 THEN
			F_ADSErrorCodeExt := 'Position out of modulo range. Position must be larger or equal to zero and less or equal to the modulo factor when using modulo positioning.';
		elsif ErrorId = 33165 Then
			F_ADSErrorCodeExt :=
				'The specified value AdditionalTurns at the Options input is not allowed. The parameter AdditionalTurns must be zero for the specified value of the parameter Direction.';
		elsif ErrorId = 33166 Then
			F_ADSErrorCodeExt :=
				'Master/Slave sync position incompatible with sync direction. The given sync positions require the slave moving in a direction which is not allowed while in synchronization phase.';
		ELSE
			F_ADSErrorCodeExt := CONCAT('ADS Error Code - ', TO_STRING(ErrorId));
		END_IF
	END_IF
END_CASE

END_FUNCTION

// Interfaces/I_Kinematic
INTERFACE I_Kinematic

METHOD Disable : BOOL
VAR_INPUT
END_VAR
END_METHOD

METHOD Enable : BOOL
VAR_INPUT
END_VAR
END_METHOD

METHOD JogCartesianAxis : BOOL
VAR_INPUT
	Axisx	 : UDINT(1..KINEMATIC_CONSTANTS.DEGREES_OF_FREEDOM_MAX);
	Forward	 : BOOL;
	Backward : BOOL;
	JogMode	 : E_JogMode;
END_VAR
END_METHOD

METHOD JogJoint : BOOL
VAR_INPUT
	Jointx	 : UDINT(1..KINEMATIC_CONSTANTS.DEGREES_OF_FREEDOM_MAX);
	Forward	 : BOOL;
	Backward : BOOL;
	JogMode	 : E_JogMode;
END_VAR
END_METHOD

METHOD Stop : BOOL
VAR_INPUT
	Deceleration : LREAL;
	Jerk		 : LREAL;
END_VAR
END_METHOD

PROPERTY ActPosition : ST_KinematicPosition
GET
END_GET
END_PROPERTY

PROPERTY Enabled : Bool
GET
END_GET
END_PROPERTY

PROPERTY InPosition : Bool
GET
END_GET
END_PROPERTY

PROPERTY Moving : Bool
GET
END_GET
END_PROPERTY

PROPERTY Override : LREAL
SET
END_SET
END_PROPERTY

PROPERTY TargetMotionParameter : REFERENCE TO ST_KinematicMotionParameter
GET
END_GET
END_PROPERTY

END_INTERFACE

// Interfaces/I_KinematicAxisRef
INTERFACE I_KinematicAxisRef

PROPERTY ACS : REFERENCE TO ARRAY[1..KINEMATIC_CONSTANTS.DEGREES_OF_FREEDOM_MAX] OF AXIS_REF
GET
END_GET
END_PROPERTY

PROPERTY DegreesOfFreedomConfigured : E_KinematicDOF
GET
END_GET
SET
END_SET
END_PROPERTY

PROPERTY MCS : REFERENCE TO ARRAY[1..KINEMATIC_CONSTANTS.DEGREES_OF_FREEDOM_MAX] OF AXIS_REF
GET
END_GET
END_PROPERTY

END_INTERFACE

// FunctionBlocks/FB_ComponentKinematicMotionAmp
FUNCTION_BLOCK FB_ComponentKinematicMotionAmp EXTENDS FB_ComponentKinematicBase IMPLEMENTS I_KinematicCm
VAR
	// Internal Variables
	_KinematicMotionAmp : FB_KinematicMotionAmpBase;
	_AmpPoints			: ARRAY[0..Parameter_Kinematic.MaxPoints] OF ST_AmpPoint;

	// HMI
	KinematicComponentAmp_HMI : ST_KinematicComponentAmp_HMI;
	_ChangeOccurred			  : BOOL;

	// Alarms
	KinematicComponentMotionAmpAlarms : ARRAY[1..KINEMATIC_COMPONENT_AMP_ALARM_COUNT] OF FB_TcAlarm;
END_VAR

VAR CONSTANT
	KINEMATIC_COMPONENT_AMP_ALARM_COUNT : UINT := 4;
END_VAR

//! @summary Initializes event function blocks using this components's name
{attribute 'call_after_online_change_slot' := '<slot>'}
METHOD PROTECTED CreateEvents
VAR
	Temp : STRING;
END_VAR

//! @description This method is called by <c>Initialize()</c> as required
Temp := CONCAT(CONCAT(CONCAT('Kinematic ', ': '), Name),
			   ' '); //Creates a utility string for alarms and other messaging that reads (example text) - "Module 10 - Main Casepacker" to be followed by the alarm or message info

F_CreateAllEventsInClass(Alarms		:= KinematicComponentMotionAmpAlarms,
						 ClassSize	:= SIZEOF(TC_EVENTS.KinematicComponentMotionAmp),
						 pInitEvent := ADR(TC_EVENTS.KinematicComponentMotionAmp.InitReferenceEvent),
						 Prefix		:= Name);

SUPER^.CreateEvents();
END_METHOD

//! @summary Provides interlocks for HMI control and updates HMI status information for this component
METHOD PROTECTED HMICommunication

//! @description This method is called cyclically by <c>CyclicLogic()</c>
SUPER^.HMICommunication();
IF NOT KinematicComponentAmp_HMI.Config.CustomOverride THEN // Custom developer is able to overrride this section via overloading HmiCommunication()
	IF ComponentBase_HMI.Status.HMIControlAvailable THEN
		IF KinematicComponentAmp_HMI.Command.BuildCmGroup THEN
			THIS^.BuildCmGroup();
			KinematicComponentAmp_HMI.Command.BuildCmGroup := FALSE;
		END_IF

		IF KinematicComponentAmp_HMI.Command.EnableCmGroup THEN
			THIS^.EnableCmGroup();
			KinematicComponentAmp_HMI.Command.EnableCmGroup := FALSE;
		END_IF

		IF KinematicComponentAmp_HMI.Command.DissolveCmGroup THEN
			THIS^.UngroupCmGroup();
			KinematicComponentAmp_HMI.Command.DissolveCmGroup := FALSE;
		END_IF

		IF KinematicComponentAmp_HMI.Command.DisableCmGroup THEN
			THIS^.DisableCmGroup();
			KinematicComponentAmp_HMI.Command.DisableCmGroup := FALSE;
		END_IF

		IF KinematicComponentAmp_HMI.Command.MoveToPointCm THEN
			THIS^.MoveToPointCartesian(KinematicComponentAmp_HMI.Command.PointSelect);
			KinematicComponentAmp_HMI.Command.MoveToPointCm := FALSE;
		END_IF

		IF KinematicComponentAmp_HMI.Command.TeachPoint THEN
			IF KinematicComponentAmp_HMI.Command.PointSelect <= Parameter_Kinematic.MaxPoints THEN
				FOR _i := 1 TO TO_UDINT(iAxis.DegreesOfFreedomConfigured) DO
					_AmpPoints[KinematicComponentAmp_HMI.Command.PointSelect].McsPosition[_i] := _ActPosition.MCS[_i];
					_AmpPoints[KinematicComponentAmp_HMI.Command.PointSelect].AcsPosition[_i] := _ActPosition.ACS[_i];
				END_FOR
			END_IF

			KinematicComponentAmp_HMI.Command.TeachPoint := FALSE;
			_ChangeOccurred								 := TRUE;
		END_IF
	END_IF

	// Status to HMI
	KinematicComponentAmp_HMI.Status.CmState := THIS^.CmState;
	IF KinematicComponentAmp_HMI.Command.PointSelect <= Parameter_Kinematic.MaxPoints THEN
		KinematicComponentAmp_HMI.Status.SelectedPoint := _AmpPoints[KinematicComponentAmp_HMI.Command.PointSelect];
	ELSE // Selection invalid
		MEMSET(ADR(KinematicComponentAmp_HMI.Status.SelectedPoint), 0, SIZEOF(KinematicComponentAmp_HMI.Status.SelectedPoint));
	END_IF
END_IF
END_METHOD

//! Provides basic error detection and event handling for this component
METHOD PROTECTED Monitoring

(*! @descriptionThis method is called cyclically by <c>CyclicLogic()</c>*)
SUPER^.Monitoring();
IF _KinematicMotionAmp.Error AND NOT _KinematicMotionAmp.InitComplete AND NOT KinematicComponentMotionAmpAlarms[E_KinematicComponentMotionAmp.CoordinatedMotionGroupInitFail].bRaised THEN
	RaiseAlarmWithStrings(Alarm := KinematicComponentMotionAmpAlarms[E_KinematicComponentMotionAmp.CoordinatedMotionGroupInitFail], F_ADSErrorCodeExt(_KinematicMotionAmp.ErrorID), '');
ELSIF NOT _KinematicMotionAmp.Error AND _KinematicMotionAmp.InitComplete AND KinematicComponentMotionAmpAlarms[E_KinematicComponentMotionAmp.CoordinatedMotionGroupInitFail].bRaised THEN
	KinematicComponentMotionAmpAlarms[E_KinematicComponentMotionAmp.CoordinatedMotionGroupInitFail].Clear(0, 0);
END_IF

IF _KinematicMotionAmp.Error AND NOT KinematicComponentMotionAmpAlarms[E_KinematicComponentMotionAmp.CoordinatedMotionGroupError].bRaised THEN
	RaiseAlarmWithStrings(Alarm := KinematicComponentMotionAmpAlarms[E_KinematicComponentMotionAmp.CoordinatedMotionGroupError], F_ADSErrorCodeExt(_KinematicMotionAmp.ErrorID), '');
ELSIF NOT _KinematicMotionAmp.Error AND KinematicComponentMotionAmpAlarms[E_KinematicComponentMotionAmp.CoordinatedMotionGroupError].bRaised THEN
	KinematicComponentMotionAmpAlarms[E_KinematicComponentMotionAmp.CoordinatedMotionGroupError].Clear(0, 0);
END_IF

_CurrentAlarmSeverity := F_GetMaxSeverityRaised(Alarms := KinematicComponentMotionAmpAlarms, CurrentSeverity := _CurrentAlarmSeverity);
END_METHOD

//! @summary Clears error flags and error IDs for this component
METHOD PUBLIC Reset : BOOL
SUPER^.Reset();
_KinematicMotionAmp.Reset();
Reset := TRUE;
END_METHOD

//! @summary This method serves as the entry point for all underlying FB logic
METHOD PUBLIC CyclicLogic
IF NOT _InitComplete THEN
	_InitComplete := Initialize();
	RETURN;
END_IF

_KinematicMotionAmp.CyclicLogic();
_Busy := SUPER^._KinematicComponentBaseBusy OR _KinematicMotionAmp.Busy;
SUPER^.CyclicLogic();
END_METHOD

PROPERTY Moving : BOOL
GET
Moving := _KinematicMotionAmp.CmState.GroupMoving OR _KinematicMotionAmp.CmState.GroupHoming OR _KinematicMotionAmp.CmState.GroupStopping;
FOR _i := 1 TO TO_UDINT(iAxis.DegreesOfFreedomConfigured) DO
	IF NOT (iAxis.ACS[_i].NcToPlc.StateDWord.2 OR iAxis.MCS[_i].NcToPlc.StateDWord.2) THEN // StatusDWord Bit 2 = Axis is logically stationary ("Axis not moving")

		// .Status.Moving is not valid if Kinematic reaches end of workspace fault
		Moving := TRUE;
	END_IF
END_FOR
END_GET
END_PROPERTY

{attribute 'monitoring' := 'variable'}
PROPERTY Override : LREAL
SET
_KinematicMotionAmp.SetOverride(Override);
SUPER^.Override := Override;
END_SET
END_PROPERTY

METHOD PUBLIC Stop : BOOL
VAR_INPUT
	Deceleration : LREAL;
	Jerk		 : LREAL;
END_VAR
IF _KinematicMotionAmp.CmState.GroupHoming OR _KinematicMotionAmp.CmState.GroupMoving OR _KinematicMotionAmp.CmState.GroupStopping OR _KinematicMotionAmp.CmState.GroupStandby THEN
	Stop := _KinematicMotionAmp.Stop(Deceleration, Jerk);
ELSE
	Stop := SUPER^.Stop(Deceleration, Jerk);
END_IF
END_METHOD

PROPERTY CmIdentAxis1 : IDENT_IN_GROUP_REF
SET
_KinematicMotionAmp.CmIdentAxis1 := CmIdentAxis1;
END_SET
END_PROPERTY

PROPERTY CmIdentAxis2 : IDENT_IN_GROUP_REF
SET
_KinematicMotionAmp.CmIdentAxis2 := CmIdentAxis2;
END_SET
END_PROPERTY

PROPERTY CmIdentAxis3 : IDENT_IN_GROUP_REF
SET
_KinematicMotionAmp.CmIdentAxis3 := CmIdentAxis3;
END_SET
END_PROPERTY

PROPERTY CmIdentAxis4 : IDENT_IN_GROUP_REF
SET
_KinematicMotionAmp.CmIdentAxis4 := CmIdentAxis4;
END_SET
END_PROPERTY

METHOD BuildCmGroup : BOOL
IF _Busy THEN
	RETURN;
END_IF

_KinematicMotionAmp.CmAxisRef REF= iAxis.MCS;
BuildCmGroup				  := _KinematicMotionAmp.BuildCmGroup();
END_METHOD

METHOD ClearPath : BOOL
ClearPath := _KinematicMotionAmp.ClearPath();
END_METHOD

{attribute 'monitoring' := 'variable'}
PROPERTY CmState : REFERENCE TO ST_KinematicComponentAmp_CmGroupState
GET
CmState REF= _KinematicMotionAmp.CmState;
END_GET
END_PROPERTY

METHOD DisableCmGroup : BOOL
IF _Busy THEN
	RETURN;
END_IF

DisableCmGroup := _KinematicMotionAmp.DisableCmGroup();
END_METHOD

METHOD EnableCmGroup : BOOL
IF _Busy THEN
	RETURN;
END_IF

EnableCmGroup := _KinematicMotionAmp.EnableCmGroup();
END_METHOD

METHOD StartMovePath : BOOL
IF _Busy THEN
	RETURN;
END_IF

StartMovePath := _KinematicMotionAmp.StartMovePath();
END_METHOD

METHOD UngroupCmGroup : BOOL
IF _Busy THEN
	RETURN;
END_IF

UngroupCmGroup := _KinematicMotionAmp.UngroupCmGroup();
END_METHOD

METHOD AddCircularMoveToPath : BOOL
VAR_INPUT
	PointIndex : UDINT;
END_VAR
IF PointIndex > Parameter_Kinematic.MaxPoints THEN
	RETURN;
END_IF

AddCircularMoveToPath := _KinematicMotionAmp.AddCircularMoveToPath(_AmpPoints[PointIndex]);
END_METHOD

METHOD AddLinearMoveToPath : BOOL
VAR_INPUT
	PointIndex : UDINT;
END_VAR
IF PointIndex > Parameter_Kinematic.MaxPoints THEN
	RETURN;
END_IF

AddLinearMoveToPath := _KinematicMotionAmp.AddLinearMoveToPath(_AmpPoints[PointIndex]);
AddLinearMoveToPath := TRUE;
END_METHOD

METHOD PUBLIC MoveToPointCartesian : BOOL
VAR_INPUT
	PointIndex : UDINT;
END_VAR
IF PointIndex > Parameter_Kinematic.MaxPoints THEN
	RETURN;
END_IF

IF _Busy THEN
	RETURN;
END_IF

IF _AmpPoints[PointIndex].CircularMove.IsCircularMove THEN
	THIS^.ClearPath();
	THIS^.AddCircularMoveToPath(PointIndex);
ELSE
	THIS^.ClearPath();
	THIS^.AddLinearMoveToPath(PointIndex);
END_IF

IF NOT _KinematicMotionAmp.Error THEN
	MoveToPointCartesian := THIS^.StartMovePath();
END_IF
END_METHOD

{attribute 'monitoring' := 'variable'}
PROPERTY PUBLIC ChangeOccurred : BOOL
GET
ChangeOccurred := _ChangeOccurred;
END_GET
SET
_ChangeOccurred := ChangeOccurred;
END_SET
END_PROPERTY

METHOD PUBLIC GetPoint : ST_AmpPoint
VAR_INPUT
	PointIndex : UDINT;
END_VAR
IF PointIndex > Parameter_Kinematic.MaxPoints THEN
	RETURN;
END_IF

GetPoint := _AmpPoints[PointIndex];
END_METHOD

{attribute 'monitoring' := 'variable'}
PROPERTY Points : REFERENCE TO ARRAY[0..Parameter_Kinematic.MaxPoints] OF ST_AmpPoint
GET
Points REF= _AmpPoints;
END_GET
END_PROPERTY

METHOD PUBLIC SetPoint : BOOL
VAR_INPUT
	Point	   : ST_AmpPoint;
	PointIndex : UDINT;
END_VAR
IF PointIndex > Parameter_Kinematic.MaxPoints THEN
	RETURN;
END_IF

_AmpPoints[PointIndex] := Point;
_ChangeOccurred		   := TRUE;
SetPoint			   := TRUE;
END_METHOD

//! @summary Basic component initialization logic
METHOD PROTECTED Initialize : BOOL;
IF SUPER^.Initialize() THEN
	IF iAxis.DegreesOfFreedomConfigured <= E_KinematicDOF.eKinematicDOF_4 THEN
		_KinematicMotionAmp.CmAxisCount := TO_UDINT(iAxis.DegreesOfFreedomConfigured);
		_KinematicMotionAmp.CyclicLogic(); // Init Run
		Initialize := _KinematicMotionAmp.InitComplete;
	ELSE
		Trace(CONCAT('Programming Error init failed with DOF in AMP FB greater than allowed - ', Name));
		RETURN;
	END_IF
END_IF
END_METHOD

END_FUNCTION_BLOCK

// Interfaces/I_KinematicCm
INTERFACE I_KinematicCm

METHOD BuildCmGroup : BOOL
END_METHOD

METHOD ClearPath : BOOL
VAR_INPUT
END_VAR
END_METHOD

METHOD DisableCmGroup : BOOL
VAR_INPUT
END_VAR
END_METHOD

METHOD EnableCmGroup : BOOL
VAR_INPUT
END_VAR
END_METHOD

METHOD StartMovePath : BOOL
VAR_INPUT
END_VAR
END_METHOD

METHOD UngroupCmGroup : BOOL
VAR_INPUT
END_VAR
END_METHOD

PROPERTY CmIdentAxis1 : IDENT_IN_GROUP_REF
SET
END_SET
END_PROPERTY

PROPERTY CmIdentAxis2 : IDENT_IN_GROUP_REF
SET
END_SET
END_PROPERTY

PROPERTY CmIdentAxis3 : IDENT_IN_GROUP_REF
SET
END_SET
END_PROPERTY

PROPERTY CmIdentAxis4 : IDENT_IN_GROUP_REF
SET
END_SET
END_PROPERTY

PROPERTY CmState : REFERENCE TO ST_KinematicComponentAmp_CmGroupState
GET
END_GET
END_PROPERTY

END_INTERFACE

// FunctionBlocks/FB_KinematicMotionAmpBase
// This Functionblock supports kinematic coordinated movement from DOF=2 to DOF=4

// Not supported are DOF=5 and DOF=6 with this FB
FUNCTION_BLOCK FB_KinematicMotionAmpBase EXTENDS FB_CyclicFB IMPLEMENTS I_KinematicCm
VAR
	// Coordinated Motion Group
	CmGroup : AXES_GROUP_REF; // link to MC Group

	// Internal Variables
	_KinematicAmpInit				 : E_InitializeState_KinematicAmp;
	_i								 : UDINT;
	_CmAxisRef						 : REFERENCE TO ARRAY[1..KINEMATIC_CONSTANTS.DEGREES_OF_FREEDOM_MAX] OF AXIS_REF;
	_AddAxisToCmGroup				 : ARRAY[1..KINEMATIC_CONSTANTS.DEGREES_OF_FREEDOM_MAX] OF MC_AddAxisToGroup;
	_GroupBuilt						 : BOOL;
	_CmIdentGroup					 : ARRAY[1..KINEMATIC_CONSTANTS.DEGREES_OF_FREEDOM_MAX] OF IDENT_IN_GROUP_REF;
	_CmAxisCount					 : UDINT := 1;
	_CmGroupReadStatus				 : MC_GroupReadStatus;
	_CmGroupState					 : ST_KinematicComponentAmp_CmGroupState;
	_UngroupAllCmAxis				 : MC_UngroupAllAxes;
	_SetOverride					 : MC_GroupSetOverride;
	_CmGroupReset					 : MC_GroupReset;
	_CmGroupEnable					 : MC_GroupEnable;
	_CmGroupDisable					 : MC_GroupDisable;
	_CmGroupStop					 : MC_GroupStop;
	_PathBuffer						 : ARRAY[1..Parameter_Kinematic.PathBufferSize] OF BYTE;
	_McPathDataRef					 : MC_PATH_DATA_REF(ADR(_PathBuffer), SIZEOF(_PathBuffer));
	_MoveLinearAbsolutePreparation	 : MC_MoveLinearAbsolutePreparation;
	_MoveCircularAbsolutePreparation : MC_MoveCircularAbsolutePreparation;
	_MovePath						 : MC_MovePath;
END_VAR

METHOD PUBLIC CyclicLogic
VAR_INPUT
END_VAR
IF NOT _InitComplete THEN
	_InitComplete := THIS^.Initialize();
	RETURN;
END_IF

_CmGroupReadStatus(AxesGroup := CmGroup, Enable := TRUE);
_CmGroupState := THIS^.MapStatus(CmGroupBuilt := _GroupBuilt);

(* Build CM Group *)
IF __ISVALIDREF(_CmAxisRef) THEN
	FOR _i := 1 TO _CmAxisCount DO
		_AddAxisToCmGroup[_i](AxesGroup := CmGroup, Axis := _CmAxisRef[_i]);
		_AddAxisToCmGroup[_i].Execute := FALSE;
	END_FOR
END_IF

FOR _i := 1 TO _CmAxisCount DO
	IF NOT _AddAxisToCmGroup[_i].Done THEN
		EXIT;
	ELSE
		_GroupBuilt := TRUE;
	END_IF
END_FOR

FOR _i := 1 TO _CmAxisCount DO
	IF _AddAxisToCmGroup[_i].Error THEN
		_GroupBuilt := FALSE;
		_Error		:= TRUE;
		_ErrorID	:= _AddAxisToCmGroup[_i].ErrorId;
		EXIT;
	END_IF
END_FOR

(* Ungroup CM Group *)
_UngroupAllCmAxis(AxesGroup := CmGroup);
IF _UngroupAllCmAxis.Error THEN
	_Error	 := TRUE;
	_ErrorID := _UngroupAllCmAxis.ErrorId;
END_IF

IF _UngroupAllCmAxis.Execute THEN
	_UngroupAllCmAxis.Execute := FALSE;
	_GroupBuilt				  := FALSE;
END_IF

(* Reset CM Group *)
_CmGroupReset(AxesGroup := CmGroup);
_CmGroupReset.Execute := FALSE;

(* Enable CM Group *)
_CmGroupEnable(AxesGroup := CmGroup);
IF _CmGroupEnable.Error THEN
	_Error	 := TRUE;
	_ErrorID := _CmGroupEnable.ErrorId;
END_IF

_CmGroupEnable.Execute := FALSE;

(* Disable CM Group *)
_CmGroupDisable(AxesGroup := CmGroup);
IF _CmGroupDisable.Error THEN
	_Error	 := TRUE;
	_ErrorID := _CmGroupDisable.ErrorId;
END_IF

_CmGroupDisable.Execute := FALSE;

(* Stop CM Group *)
_CmGroupStop(AxesGroup := CmGroup);
IF _CmGroupStop.Error THEN
	_Error	 := TRUE;
	_ErrorID := _CmGroupStop.ErrorId;
END_IF

_CmGroupStop.Execute := FALSE;

(* Move CM Group *)
_MovePath(AxesGroup := CmGroup, PathData := _McPathDataRef);
IF _MovePath.Error THEN
	_Error	 := TRUE;
	_ErrorID := _MovePath.ErrorId;
END_IF

_MovePath.Execute := FALSE;

(* Map Error from Group *)
IF NOT _Error THEN
	_Error	 := _CmGroupState.Error;
	_ErrorId := _CmGroupState.ErrorId;
END_IF

(* Busy monitoring *)
_Busy := _UngroupAllCmAxis.Busy OR _CmGroupState.GroupMoving OR _CmGroupState.GroupHoming OR _CmGroupState.GroupStopping OR _CmGroupDisable.Busy OR _CmGroupEnable.Busy OR _CmGroupStop.Busy;
IF NOT _Busy THEN
	FOR _i := 1 TO _CmAxisCount DO
		IF _AddAxisToCmGroup[_i].Busy THEN
			_Busy := TRUE;
			EXIT;
		END_IF
	END_FOR
END_IF
END_METHOD

METHOD PUBLIC BuildCmGroup : BOOL
BuildCmGroup := FALSE;
IF NOT __ISVALIDREF(_CmAxisRef) THEN
	TRACE('Add Axis to Group - Axis Reference to add not set in AxisRef Property!');
	RETURN;
END_IF

IF _Busy THEN
	RETURN;
END_IF

FOR _i := 1 TO _CmAxisCount DO
	_AddAxisToCmGroup[_i].IdentInGroup := _CmIdentGroup[_i];
	_AddAxisToCmGroup[_i].Execute	   := TRUE;
END_FOR

BuildCmGroup := TRUE;
END_METHOD

METHOD ClearPath : BOOL
_McPathDataRef.ClearPath();
ClearPath := TRUE;
END_METHOD

METHOD DisableCmGroup : BOOL
IF _Busy THEN
	RETURN;
END_IF

_CmGroupDisable.Execute := TRUE;
DisableCmGroup			:= TRUE;
END_METHOD

METHOD EnableCmGroup : BOOL
IF _Busy THEN
	RETURN;
END_IF

_CmGroupEnable.Execute := TRUE;
EnableCmGroup		   := TRUE;
END_METHOD

METHOD StartMovePath : BOOL
IF _Busy THEN
	RETURN;
END_IF

_MovePath.Execute := TRUE;
StartMovePath	  := TRUE;
END_METHOD

METHOD UngroupCmGroup : BOOL
IF _Busy THEN
	RETURN;
END_IF

_UngroupAllCmAxis.Execute := TRUE;
UngroupCmGroup			  := TRUE;
END_METHOD

PROPERTY CmIdentAxis1 : IDENT_IN_GROUP_REF
SET
_CmIdentGroup[1] := CmIdentAxis1;
END_SET
END_PROPERTY

PROPERTY CmIdentAxis2 : IDENT_IN_GROUP_REF
SET
_CmIdentGroup[2] := CmIdentAxis2;
END_SET
END_PROPERTY

PROPERTY CmIdentAxis3 : IDENT_IN_GROUP_REF
SET
_CmIdentGroup[3] := CmIdentAxis3;
END_SET
END_PROPERTY

PROPERTY CmIdentAxis4 : IDENT_IN_GROUP_REF
SET
_CmIdentGroup[4] := CmIdentAxis4;
END_SET
END_PROPERTY

{attribute 'monitoring' := 'variable'}
PROPERTY CmState : REFERENCE TO ST_KinematicComponentAmp_CmGroupState
GET
CmState REF= _CmGroupState;
END_GET
END_PROPERTY

METHOD AddCircularMoveToPath : BOOL
VAR_INPUT
	AmpPoint : REFERENCE TO ST_AmpPoint;
END_VAR
IF NOT __ISVALIDREF(AmpPoint) THEN
	RETURN;
END_IF

_MoveCircularAbsolutePreparation(PathData				  := _McPathDataRef,
								 CircMode				  := AmpPoint.CircularMove.CircMode,
								 AuxPoint				  := ADR(AmpPoint.CircularMove.AuxPoint),
								 AuxPointCount			  := 3,
								 EndPoint				  := ADR(AmpPoint.McsPosition),
								 EndPointCount			  := _CmAxisCount,
								 PathChoice				  := AmpPoint.CircularMove.PathChoice,
								 Velocity				  := AmpPoint.Velocity,
								 Acceleration			  := AmpPoint.Acceleration,
								 Deceleration			  := AmpPoint.Deceleration,
								 Jerk					  := AmpPoint.Jerk,
								 BufferMode				  := AmpPoint.BufferMode,
								 TransitionMode			  := AmpPoint.TransitionMode,
								 TransitionParameter	  := ADR(AmpPoint.TransitionParameter),
								 TransitionParameterCount := AmpPoint.TransitionParameterCount,
								 InvokeId				  := AmpPoint.InvokeId,
								 Error					  => _Error,
								 ErrorId				  => _ErrorId);

AddCircularMoveToPath := TRUE;
END_METHOD

METHOD AddLinearMoveToPath : BOOL
VAR_INPUT
	AmpPoint : REFERENCE TO ST_AmpPoint;
END_VAR
IF NOT __ISVALIDREF(AmpPoint) THEN
	RETURN;
END_IF

_MoveLinearAbsolutePreparation(PathData					:= _McPathDataRef,
							   Position					:= ADR(AmpPoint.McsPosition),
							   PositionCount			:= _CmAxisCount,
							   Velocity					:= AmpPoint.Velocity,
							   Acceleration				:= AmpPoint.Acceleration,
							   Deceleration				:= AmpPoint.Deceleration,
							   Jerk						:= AmpPoint.Jerk,
							   BufferMode				:= AmpPoint.BufferMode,
							   TransitionMode			:= AmpPoint.TransitionMode,
							   TransitionParameter		:= ADR(AmpPoint.TransitionParameter),
							   TransitionParameterCount := AmpPoint.TransitionParameterCount,
							   InvokeId					:= AmpPoint.InvokeId,
							   Error					=> _Error,
							   ErrorId					=> _ErrorId);

AddLinearMoveToPath := TRUE;
END_METHOD

METHOD PRIVATE MapStatus : ST_KinematicComponentAmp_CmGroupState
VAR_INPUT
	CmGroupBuilt : BOOL;
END_VAR
MapStatus.GroupBuilt	   := CmGroupBuilt;
MapStatus.GroupMoving	   := _CmGroupReadStatus.GroupMoving;
MapStatus.GroupHoming	   := _CmGroupReadStatus.GroupHoming;
MapStatus.GroupErrorStop   := _CmGroupReadStatus.GroupErrorStop;
MapStatus.GroupNotReady	   := _CmGroupReadStatus.GroupNotReady;
MapStatus.GroupStandby	   := _CmGroupReadStatus.GroupStandby;
MapStatus.GroupStopping	   := _CmGroupReadStatus.GroupStopping;
MapStatus.GroupDisabled	   := _CmGroupReadStatus.GroupDisabled;
MapStatus.AllAxesStanding  := _CmGroupReadStatus.AllAxesStanding;
MapStatus.ConstantVelocity := _CmGroupReadStatus.ConstantVelocity;
MapStatus.Accelerating	   := _CmGroupReadStatus.Accelerating;
MapStatus.Decelerating	   := _CmGroupReadStatus.Decelerating;
MapStatus.InPosition	   := _CmGroupReadStatus.InPosition;
MapStatus.Error			   := _CmGroupReadStatus.Error;
MapStatus.ErrorId		   := _CmGroupReadStatus.ErrorId;
END_METHOD

METHOD PUBLIC Reset : BOOL
VAR_INPUT
END_VAR
_CmGroupReset.Execute := TRUE;
_Error				  := FALSE;
_ErrorId			  := 0;
Reset				  := TRUE;
END_METHOD

METHOD PUBLIC SetOverride : BOOL
VAR_INPUT
	Override : MC_LREAL := 100.0; // 100.0 = 100% Full Speed
END_VAR
Override := Override / 100.0;
_SetOverride(AxesGroup := CmGroup, Enable := TRUE, VelFactor := Override);
SetOverride := TRUE;
END_METHOD

METHOD PUBLIC Stop : BOOL
VAR_INPUT
	Deceleration : LREAL;
	Jerk		 : LREAL;
END_VAR
IF Deceleration = 0 OR Jerk = 0 THEN
	_CmGroupStop.Deceleration := Parameter_Kinematic.DefaultStopDeceleration;
	_CmGroupStop.Jerk		  := Parameter_Kinematic.DefaultStopDecelerationJerk;
ELSE
	_CmGroupStop.Deceleration := Deceleration;
	_CmGroupStop.Jerk		  := Jerk;
END_IF

_CmGroupStop.Execute := TRUE;
Stop				 := TRUE;
END_METHOD

{attribute 'monitoring' := 'variable'}
PROPERTY Public CmAxisCount : UDINT
SET
_CmAxisCount := CmAxisCount;
END_SET
END_PROPERTY

{attribute 'monitoring' := 'variable'}
PROPERTY PUBLIC CmAxisRef : REFERENCE TO ARRAY[1..KINEMATIC_CONSTANTS.DEGREES_OF_FREEDOM_MAX] OF AXIS_REF
GET
CmAxisRef Ref= _CmAxisRef;
END_GET
SET
_CmAxisRef REF= CmAxisRef;
END_SET
END_PROPERTY

METHOD PROTECTED Initialize : BOOL
VAR_INPUT
END_VAR
CASE _KinematicAmpInit OF
	E_InitializeState_KinematicAmp.eInitializeState_Start:
		Initialize := FALSE;
		IF _CmAxisCount > 4 THEN
			TRACE('Too many Axes connected to AMP FB! Only up to DOF=4 possible!');
			_KinematicAmpInit := E_InitializeState_KinematicAmp.eInitializeState_Failed;
			RETURN;
		ELSE
			_KinematicAmpInit := E_InitializeState_KinematicAmp.eInitializeState_CheckLinking;
		END_IF

	E_InitializeState_KinematicAmp.eInitializeState_CheckLinking:
		IF F_GetMappingStatus(ADR(CmGroup.NcToPlc), SIZEOF(CmGroup.NcToPlc)) <> EPlcMappingStatus.MS_Mapped OR
		   F_GetMappingStatus(ADR(CmGroup.PlcToNc), SIZEOF(CmGroup.PlcToNc)) <> EPlcMappingStatus.MS_Mapped THEN
			Trace('Programming Error init failed with Group Link missing!');
			_KinematicAmpInit := E_InitializeState_KinematicAmp.eInitializeState_Failed;
		ELSE
			_KinematicAmpInit := E_InitializeState_KinematicAmp.eInitializeState_Done;
		END_IF

	E_InitializeState_KinematicAmp.eInitializeState_Done:
		_Busy	   := FALSE;
		Initialize := TRUE;

	E_InitializeState_KinematicAmp.eInitializeState_Failed:
		_Busy  := FALSE;
		_Error := TRUE;
END_CASE
END_METHOD

END_FUNCTION_BLOCK

// FunctionBlocks/FB_ComponentKinematicMotionCamming
FUNCTION_BLOCK FB_ComponentKinematicMotionCamming EXTENDS FB_ComponentKinematicBase IMPLEMENTS I_KinematicCamming
VAR
	// Internal Variables
	_AcsAxesCam : FB_KinematicCamming;
	_McsAxesCam : FB_KinematicCamming;
	_CamPoints	: ARRAY[0..Parameter_Kinematic.MaxPoints] OF ST_BasePoint;

	// HMI
	KinematicComponentCam_HMI : ST_KinematicComponentCam_HMI;
	_ChangeOccurred			  : BOOL;

	// Alarms
	KinematicComponentMotionCamAlarms : ARRAY[1..KINEMATIC_COMPONENT_CAM_ALARM_COUNT] OF FB_TcAlarm;
END_VAR

VAR CONSTANT
	KINEMATIC_COMPONENT_CAM_ALARM_COUNT : UINT := 3;
END_VAR

//! @summary Initializes event function blocks using this components's name
{attribute 'call_after_online_change_slot' := '<slot>'}
METHOD PROTECTED CreateEvents
VAR
	Temp : STRING;
END_VAR

//! @description This method is called by <c>Initialize()</c> as required
Temp := CONCAT(CONCAT(CONCAT('Kinematic ', ': '), Name),
			   ' '); //Creates a utility string for alarms and other messaging that reads (example text) - "Module 10 - Main Casepacker" to be followed by the alarm or message info

F_CreateAllEventsInClass(Alarms		:= KinematicComponentMotionCamAlarms,
						 ClassSize	:= SIZEOF(TC_EVENTS.KinematicComponentMotionCam),
						 pInitEvent := ADR(TC_EVENTS.KinematicComponentMotionCam.InitReferenceEvent),
						 Prefix		:= Name);

SUPER^.CreateEvents();
END_METHOD

//! @summary Provides interlocks for HMI control and updates HMI status information for this component
METHOD PROTECTED HMICommunication
VAR
	_TempPointVelocity	   : ARRAY[1..KINEMATIC_CONSTANTS.DEGREES_OF_FREEDOM_MAX] OF LREAL;
	_TempPointAcceleration : ARRAY[1..KINEMATIC_CONSTANTS.DEGREES_OF_FREEDOM_MAX] OF LREAL;
	_TempPointJerk		   : ARRAY[1..KINEMATIC_CONSTANTS.DEGREES_OF_FREEDOM_MAX] OF LREAL;
END_VAR

VAR_INST
	// Test - to be deleted
	AddPointToPath : BOOL;
	CamIn		   : BOOL;
	StartMovePath  : BOOL;
	CamOut		   : BOOL;
	DeletePath	   : BOOL;
END_VAR
SUPER^.HMICommunication();
IF NOT KinematicComponentCam_HMI.Config.CustomOverride THEN // Custom developer is able to overrride this section via overloading HmiCommunication()
	IF ComponentBase_HMI.Status.HMIControlAvailable THEN
		IF KinematicComponentCam_HMI.Command.MoveToPointCam THEN
			KinematicComponentCam_HMI.Command.MoveToPointCam := FALSE;
			THIS^.CamStartMovePath(TargetMoveVelocity	  := Parameter_Kinematic.CamDefaultMoveVelocity,
								   TargetMoveAcceleration := Parameter_Kinematic.CamDefaultMoveAcceleration,
								   TargetMoveDeceleration := Parameter_Kinematic.CamDefaultMoveDeceleration,
								   TargetMoveJerk		  := Parameter_Kinematic.CamDefaultMoveJerk);
		END_IF

		IF KinematicComponentCam_HMI.Command.CamAddPoint THEN
			KinematicComponentCam_HMI.Command.CamAddPoint := FALSE;
			IF KinematicComponentCam_HMI.Command.PointSelect <= Parameter_Kinematic.MaxPoints THEN
				THIS^.CamAddPointToPath(MotionFunctionFirstPoint := MC_MotionFunctionType.MOTIONFUNCTYPE_POLYNOM5,
										MotionFunctionThisPoint	 := MC_MotionFunctionType.MOTIONFUNCTYPE_POLYNOM5,
										PointNumber				 := 2,
										TotalPointsInTable		 := 2,
										PointIndex				 := KinematicComponentCam_HMI.Command.PointSelect,
										PointVelocity			 := _TempPointVelocity, // Vel in each point is 0, HMI is move to one point only!
										PointAcceleration		 := _TempPointAcceleration,
										PointJerk				 := _TempPointJerk);
			END_IF
		END_IF

		IF KinematicComponentCam_HMI.Command.CamIn THEN
			KinematicComponentCam_HMI.Command.CamIn := FALSE;
			THIS^.CamIn();
		END_IF

		IF KinematicComponentCam_HMI.Command.CamOut THEN
			KinematicComponentCam_HMI.Command.CamOut := FALSE;
			THIS^.CamOut();
		END_IF

		IF KinematicComponentCam_HMI.Command.CamDeletePoint THEN
			KinematicComponentCam_HMI.Command.CamDeletePoint := FALSE;
			THIS^.CamClearPath();
		END_IF

		IF KinematicComponentCam_HMI.Command.TeachPoint THEN
			IF KinematicComponentCam_HMI.Command.PointSelect <= Parameter_Kinematic.MaxPoints THEN
				FOR _i := 1 TO TO_UDINT(iAxis.DegreesOfFreedomConfigured) DO
					_CamPoints[KinematicComponentCam_HMI.Command.PointSelect].McsPosition[_i] := _ActPosition.MCS[_i];
					_CamPoints[KinematicComponentCam_HMI.Command.PointSelect].AcsPosition[_i] := _ActPosition.ACS[_i];
				END_FOR
			END_IF

			KinematicComponentCam_HMI.Command.TeachPoint := FALSE;
			_ChangeOccurred								 := TRUE;
		END_IF
	END_IF

	// Status to HMI
	KinematicComponentCam_HMI.Status.CammingActive := THIS^.CammingActive;
	IF KinematicComponentCam_HMI.Command.PointSelect <= Parameter_Kinematic.MaxPoints THEN
		KinematicComponentCam_HMI.Status.SelectedPoint := _CamPoints[KinematicComponentCam_HMI.Command.PointSelect];
	ELSE // Selection invalid
		MEMSET(ADR(KinematicComponentCam_HMI.Status.SelectedPoint), 0, SIZEOF(KinematicComponentCam_HMI.Status.SelectedPoint));
	END_IF
END_IF
END_METHOD

//! Provides basic error detection and event handling for this component
METHOD PROTECTED Monitoring

(*! @descriptionThis method is called cyclically by <c>CyclicLogic()</c>*)
SUPER^.Monitoring();
IF _AcsAxesCam.Error AND NOT KinematicComponentMotionCamAlarms[E_KinematicComponentMotionCam.CammingMotionAcsAxes].bRaised THEN
	RaiseAlarmWithStrings(Alarm := KinematicComponentMotionCamAlarms[E_KinematicComponentMotionCam.CammingMotionAcsAxes], F_ADSErrorCodeExt(_AcsAxesCam.ErrorID), '');
ELSIF NOT _AcsAxesCam.Error AND KinematicComponentMotionCamAlarms[E_KinematicComponentMotionCam.CammingMotionAcsAxes].bRaised THEN
	KinematicComponentMotionCamAlarms[E_KinematicComponentMotionCam.CammingMotionAcsAxes].Clear(0, 0);
END_IF

IF _McsAxesCam.Error AND NOT KinematicComponentMotionCamAlarms[E_KinematicComponentMotionCam.CammingMotionMcsAxes].bRaised THEN
	RaiseAlarmWithStrings(Alarm := KinematicComponentMotionCamAlarms[E_KinematicComponentMotionCam.CammingMotionMcsAxes], F_ADSErrorCodeExt(_McsAxesCam.ErrorID), '');
ELSIF NOT _McsAxesCam.Error AND KinematicComponentMotionCamAlarms[E_KinematicComponentMotionCam.CammingMotionMcsAxes].bRaised THEN
	KinematicComponentMotionCamAlarms[E_KinematicComponentMotionCam.CammingMotionMcsAxes].Clear(0, 0);
END_IF

_CurrentAlarmSeverity := F_GetMaxSeverityRaised(Alarms := KinematicComponentMotionCamAlarms, CurrentSeverity := _CurrentAlarmSeverity);
END_METHOD

//! @summary Clears error flags and error IDs for this component
METHOD PUBLIC Reset : BOOL
_AcsAxesCam.Reset();
_McsAxesCam.Reset();
IF (NOT _AcsAxesCam.CammingActive AND NOT _McsAxesCam.CammingActive) OR (SUPER^._McPowerAcsErrorActive OR SUPER^._McPowerMcsErrorActive) THEN
	Reset := SUPER^.Reset();
ELSE
	_Error	 := FALSE;
	_ErrorId := 0;
	Reset	 := TRUE;
END_IF
END_METHOD

//! @summary This method serves as the entry point for all underlying FB logic
METHOD PUBLIC CyclicLogic
IF NOT _InitComplete THEN
	_InitComplete := Initialize();
	RETURN;
END_IF

(* Cyclic Call of Axis Ref to Camming *)
_AcsAxesCam.CamAxisCount := TO_UDINT(iAxis.DegreesOfFreedomConfigured);
_AcsAxesCam.CamAxisRef	 REF= iAxis.ACS;
_McsAxesCam.CamAxisCount := TO_UDINT(iAxis.DegreesOfFreedomConfigured);
_McsAxesCam.CamAxisRef	 REF= iAxis.MCS;

(* Camming for ACS/Joint Axes *)
_AcsAxesCam.CyclicLogic();
IF _AcsAxesCam.Error THEN
	_Error	 := TRUE;
	_ErrorId := _AcsAxesCam.ErrorID;
END_IF

(* Camming for Mcs/Cartesian Axes *)
_McsAxesCam.CyclicLogic();
IF _McsAxesCam.Error THEN
	_Error	 := TRUE;
	_ErrorId := _McsAxesCam.ErrorID;
END_IF

(* Cam Out in Error or Disabled State *)
IF _Error OR NOT Enabled THEN
	THIS^.CamOut();
END_IF

_Busy := THIS^._KinematicComponentBaseBusy OR _AcsAxesCam.Busy OR _McsAxesCam.Busy;
SUPER^.CyclicLogic();
END_METHOD

METHOD PUBLIC Disable : BOOL
_AcsAxesCam.Disable();
_McsAxesCam.Disable();
Disable := Super^.Disable();
END_METHOD

METHOD PUBLIC Enable : BOOL
_AcsAxesCam.Enable();
_McsAxesCam.Enable();
Enable := Super^.Enable();
END_METHOD

{attribute 'monitoring' := 'variable'}
PROPERTY Override : LREAL
SET
_AcsAxesCam.SetOverride(Override);
_McsAxesCam.SetOverride(Override);
SUPER^.Override := Override;
END_SET
END_PROPERTY

METHOD PUBLIC Stop : BOOL
VAR_INPUT
	Deceleration : LREAL;
	Jerk		 : LREAL;
END_VAR
IF _McsAxesCam.CammingActive THEN
	Stop := _McsAxesCam.Stop(Deceleration, Jerk);
ELSIF _AcsAxesCam.CammingActive THEN
	Stop := _AcsAxesCam.Stop(Deceleration, Jerk);
ELSE
	Stop := SUPER^.Stop(Deceleration, Jerk);
END_IF
END_METHOD

METHOD CamClearPath : BOOL
IF _Busy THEN
	RETURN;
END_IF

IF NOT _McsAxesCam.CammingActive THEN
	CamClearPath := _McsAxesCam.CamClearPath();
END_IF

IF NOT _AcsAxesCam.CammingActive THEN
	CamClearPath := _AcsAxesCam.CamClearPath();
END_IF
END_METHOD

METHOD CamIn : BOOL
IF _Busy THEN
	RETURN;
END_IF

IF SUPER^.KinematicStatus = E_KinStatus.KinStatus_Empty AND NOT _McsAxesCam.CammingActive THEN
	CamIn := _AcsAxesCam.CamIn();
ELSIF SUPER^.KinematicStatus = E_KinStatus.KinStatus_Ready AND NOT _AcsAxesCam.CammingActive THEN
	CamIn := _McsAxesCam.CamIn();
ELSE
	CamIn := FALSE;
END_IF
END_METHOD

{attribute 'monitoring' := 'variable'}
PROPERTY CammingActive : BOOL
GET
CammingActive := _McsAxesCam.CammingActive OR _AcsAxesCam.CammingActive;
END_GET
END_PROPERTY

METHOD CamOut : BOOL
IF _Busy THEN
	RETURN;
END_IF

IF _AcsAxesCam.CammingActive THEN
	CamOut := _AcsAxesCam.CamOut();
ELSIF _McsAxesCam.CammingActive THEN
	CamOut := _McsAxesCam.CamOut();
ELSE
	CamOut := FALSE;
END_IF
END_METHOD

METHOD CamStartMovePath : BOOL
VAR_INPUT
	TargetMoveVelocity	   : LREAL := Parameter_Kinematic.CamDefaultMoveVelocity;	  // Move Velocity for Cam Table Master !!!Needs to consider all Slave dynamics, all Slaves try to follow Master setpoints!!!
	TargetMoveAcceleration : LREAL := Parameter_Kinematic.CamDefaultMoveAcceleration; // Move Acceleration for Cam Table Master !!!Needs to consider all Slave dynamics, all Slaves try to follow Master setpoints!!!
	TargetMoveDeceleration : LREAL := Parameter_Kinematic.CamDefaultMoveDeceleration; // Move Deceleration for Cam Table Master !!!Needs to consider all Slave dynamics, all Slaves try to follow Master setpoints!!!
	TargetMoveJerk		   : LREAL := Parameter_Kinematic.CamDefaultMoveJerk;		  // Move Jerk for Cam Table Master !!!Needs to consider all Slave dynamics, all Slaves try to follow Master setpoints!!!
END_VAR
IF _Busy THEN
	RETURN;
END_IF

IF SUPER^.KinematicStatus = E_KinStatus.KinStatus_Empty AND _AcsAxesCam.CammingActive THEN
	CamStartMovePath := _AcsAxesCam.CamStartMovePath(TargetMoveVelocity		:= TargetMoveVelocity,
													 TargetMoveAcceleration := TargetMoveAcceleration,
													 TargetMoveDeceleration := TargetMoveDeceleration,
													 TargetMoveJerk			:= TargetMoveJerk);
ELSIF SUPER^.KinematicStatus = E_KinStatus.KinStatus_Ready AND _McsAxesCam.CammingActive THEN
	CamStartMovePath := _McsAxesCam.CamStartMovePath(TargetMoveVelocity		:= TargetMoveVelocity,
													 TargetMoveAcceleration := TargetMoveAcceleration,
													 TargetMoveDeceleration := TargetMoveDeceleration,
													 TargetMoveJerk			:= TargetMoveJerk);
ELSE
	CamStartMovePath := FALSE;
END_IF
END_METHOD

METHOD PUBLIC BuildKinGroup : BOOL
IF _McsAxesCam.CammingActive OR _AcsAxesCam.CammingActive THEN
	RETURN;
END_IF

BuildKinGroup := SUPER^.BuildKinGroup();
END_METHOD

METHOD PUBLIC DissolveKinGroup : BOOL
IF _McsAxesCam.CammingActive OR _AcsAxesCam.CammingActive THEN
	RETURN;
END_IF

DissolveKinGroup := SUPER^.DissolveKinGroup();
END_METHOD

METHOD CamAddPointToPath : BOOL
VAR_INPUT
	MotionFunctionFirstPoint : MC_MotionFunctionType;										  // Motion Function Type of initial Point in Cam Table. Start Postion is defined by current Positon of Axes.
	MotionFunctionThisPoint	 : MC_MotionFunctionType;										  // Motion Function Type of this Point to be added to Cam-Table
	PointNumber				 : UDINT(2..Parameter_Kinematic.MaxCammingPositionsPerTable);	  // Number of Point to be added to Cam Table, must be strictly increasing without gaps
	TotalPointsInTable		 : UDINT(2..Parameter_Kinematic.MaxCammingPositionsPerTable);	  // Total Number of Points in final Cam Table
	PointVelocity			 : ARRAY[1..KINEMATIC_CONSTANTS.DEGREES_OF_FREEDOM_MAX] OF LREAL; // Slave Velocity at this Point in Cam Table
	PointAcceleration		 : ARRAY[1..KINEMATIC_CONSTANTS.DEGREES_OF_FREEDOM_MAX] OF LREAL; // Slave Acceleration at this Point in Cam Table
	PointJerk				 : ARRAY[1..KINEMATIC_CONSTANTS.DEGREES_OF_FREEDOM_MAX] OF LREAL; // Slave Jerk at this Point in Cam Table
	PointIndex				 : UDINT;														  // Index of Point in structure of ST_BasePoint
END_VAR
IF _AcsAxesCam.CammingActive OR _McsAxesCam.CammingActive OR _AcsAxesCam.Busy OR _McsAxesCam.Busy THEN
	RETURN;
END_IF

IF SUPER^.KinematicStatus = E_KinStatus.KinStatus_Empty THEN
	CamAddPointToPath := _AcsAxesCam.CamAddPointToPath(MotionFunctionFirstPoint := MotionFunctionFirstPoint,
													   MotionFunctionThisPoint	:= MotionFunctionThisPoint,
													   PointNumber				:= PointNumber,
													   TotalPointsInTable		:= TotalPointsInTable,
													   Point					:= _CamPoints[PointIndex].AcsPosition,
													   PointVelocity			:= PointVelocity,
													   PointAcceleration		:= PointAcceleration,
													   PointJerk				:= PointJerk);
ELSIF SUPER^.KinematicStatus = E_KinStatus.KinStatus_Ready THEN
	CamAddPointToPath := _McsAxesCam.CamAddPointToPath(MotionFunctionFirstPoint := MotionFunctionFirstPoint,
													   MotionFunctionThisPoint	:= MotionFunctionThisPoint,
													   PointNumber				:= PointNumber,
													   TotalPointsInTable		:= TotalPointsInTable,
													   Point					:= _CamPoints[PointIndex].McsPosition,
													   PointVelocity			:= PointVelocity,
													   PointAcceleration		:= PointAcceleration,
													   PointJerk				:= PointJerk);
ELSE
	CamAddPointToPath := FALSE;
END_IF
END_METHOD

PROPERTY PUBLIC ChangeOccurred : BOOL
GET
ChangeOccurred := _ChangeOccurred;
END_GET
SET
_ChangeOccurred := ChangeOccurred;
END_SET
END_PROPERTY

METHOD PUBLIC GetPoint : ST_BasePoint
VAR_INPUT
	PointIndex : UDINT;
END_VAR
IF PointIndex > Parameter_Kinematic.MaxPoints THEN
	RETURN;
END_IF

GetPoint := _CamPoints[PointIndex];
END_METHOD

PROPERTY Points : REFERENCE TO ARRAY[0..Parameter_Kinematic.MaxPoints] OF ST_BasePoint
GET
Points REF= _CamPoints;
END_GET
END_PROPERTY

METHOD PUBLIC SetPoint : BOOL
VAR_INPUT
	Point	   : ST_BasePoint;
	PointIndex : UDINT;
END_VAR
IF PointIndex > Parameter_Kinematic.MaxPoints THEN
	RETURN;
END_IF

_CamPoints[PointIndex] := Point;
_ChangeOccurred		   := TRUE;
SetPoint			   := TRUE;
END_METHOD

//! @summary Basic component initialization logic
METHOD PROTECTED Initialize : BOOL;
_AcsAxesCam.CamAxisCount := TO_UDINT(iAxis.DegreesOfFreedomConfigured);
_AcsAxesCam.CamAxisRef	 REF= iAxis.ACS;
_McsAxesCam.CamAxisCount := TO_UDINT(iAxis.DegreesOfFreedomConfigured);
_McsAxesCam.CamAxisRef	 REF= iAxis.MCS;
_AcsAxesCam.CyclicLogic(); // Init Run
_McsAxesCam.CyclicLogic(); // Init Run
IF SUPER^.Initialize() THEN
	Initialize := _AcsAxesCam.InitComplete AND _McsAxesCam.InitComplete;
END_IF
END_METHOD

END_FUNCTION_BLOCK

// Interfaces/I_KinematicCamming
INTERFACE I_KinematicCamming

METHOD CamClearPath : BOOL
VAR_INPUT
END_VAR
END_METHOD

METHOD CamIn : BOOL
VAR_INPUT
END_VAR
END_METHOD

METHOD CamOut : BOOL
VAR_INPUT
END_VAR
END_METHOD

METHOD CamStartMovePath : BOOL
VAR_INPUT
	TargetMoveVelocity	   : LREAL := Parameter_Kinematic.CamDefaultMoveVelocity;	  // Move Velocity for Cam Table Master !!!Needs to consider all Slave dynamics, all Slaves try to follow Master setpoints!!!
	TargetMoveAcceleration : LREAL := Parameter_Kinematic.CamDefaultMoveAcceleration; // Move Acceleration for Cam Table Master !!!Needs to consider all Slave dynamics, all Slaves try to follow Master setpoints!!!
	TargetMoveDeceleration : LREAL := Parameter_Kinematic.CamDefaultMoveDeceleration; // Move Deceleration for Cam Table Master !!!Needs to consider all Slave dynamics, all Slaves try to follow Master setpoints!!!
	TargetMoveJerk		   : LREAL := Parameter_Kinematic.CamDefaultMoveJerk;		  // Move Jerk for Cam Table Master !!!Needs to consider all Slave dynamics, all Slaves try to follow Master setpoints!!!
END_VAR
END_METHOD

PROPERTY CammingActive : BOOL
GET
END_GET
END_PROPERTY

END_INTERFACE

// FunctionBlocks/FB_KinematicCamming
FUNCTION_BLOCK FB_KinematicCamming EXTENDS FB_CyclicFB IMPLEMENTS I_KinematicCamming
VAR
	// Kinematic Axis
	_CamVirtualMaster	  : AXIS_REF;
	_CamAxisRef			  : REFERENCE TO ARRAY[1..KINEMATIC_CONSTANTS.DEGREES_OF_FREEDOM_MAX] OF AXIS_REF;
	_CamAxisCount		  : UDINT													  := 1;
	_MotionFunctionPoints : UDINT(2..Parameter_Kinematic.MaxCammingPositionsPerTable) := 2;

	// Camming
	_McCamTableSelect		   : ARRAY[1..KINEMATIC_CONSTANTS.DEGREES_OF_FREEDOM_MAX] OF MC_CamTableSelect;
	_TableCamRef			   : ARRAY[1..KINEMATIC_CONSTANTS.DEGREES_OF_FREEDOM_MAX] OF MC_CAM_REF;
	_MotionFunctionPointsAxis1 : ARRAY[1..Parameter_Kinematic.MaxCammingPositionsPerTable] OF MC_MotionFunctionPoint;
	_MotionFunctionPointsAxis2 : ARRAY[1..Parameter_Kinematic.MaxCammingPositionsPerTable] OF MC_MotionFunctionPoint;
	_MotionFunctionPointsAxis3 : ARRAY[1..Parameter_Kinematic.MaxCammingPositionsPerTable] OF MC_MotionFunctionPoint;
	_MotionFunctionPointsAxis4 : ARRAY[1..Parameter_Kinematic.MaxCammingPositionsPerTable] OF MC_MotionFunctionPoint;
	_MotionFunctionPointsAxis5 : ARRAY[1..Parameter_Kinematic.MaxCammingPositionsPerTable] OF MC_MotionFunctionPoint;
	_MotionFunctionPointsAxis6 : ARRAY[1..Parameter_Kinematic.MaxCammingPositionsPerTable] OF MC_MotionFunctionPoint;
	_McCamIn				   : ARRAY[1..KINEMATIC_CONSTANTS.DEGREES_OF_FREEDOM_MAX] OF MC_CamIn;
	_McCamOut				   : ARRAY[1..KINEMATIC_CONSTANTS.DEGREES_OF_FREEDOM_MAX] OF MC_CamOut;
	_McPowerVirtualMaster	   : MC_POWER;
	_McMoveAbs				   : MC_MoveAbsolute;
	_McHalt					   : MC_Halt;
	_McReset				   : MC_Reset;

	// Internal Variables
	_KinematicCamInit		  : E_InitializeState_KinematicCamming := E_InitializeState_KinematicCamming.eInitializeState_Start;
	_i						  : UDINT;
	_MotionFunctionFirstPoint : MC_MotionFunctionType := MC_MotionFunctionType.MOTIONFUNCTYPE_POLYNOM5;
END_VAR

METHOD PUBLIC CyclicLogic
IF NOT _InitComplete THEN
	_InitComplete := THIS^.Initialize();
	RETURN;
END_IF

(* Power Virtual Master *)
_McPowerVirtualMaster(Axis := _CamVirtualMaster, Enable_Positive := TRUE, Enable_Negative := TRUE);
IF _McPowerVirtualMaster.Error THEN
	_Error	 := TRUE;
	_ErrorId := _McPowerVirtualMaster.ErrorID;
END_IF

(* Reset Virtual Master *)
_McReset(Axis := _CamVirtualMaster);
IF _McReset.Error THEN
	_Error	 := TRUE;
	_ErrorId := _McReset.ErrorID;
END_IF

_McReset.Execute := FALSE;

(* Stop Virtual Master *)
_McHalt(Axis := _CamVirtualMaster);
IF _McHalt.Error THEN
	_Error	 := TRUE;
	_ErrorId := _McHalt.ErrorID;
END_IF

_McHalt.Execute := FALSE;

(* Move Virtual Master *)
_McMoveAbs(Axis := _CamVirtualMaster);
IF _McMoveAbs.Error THEN
	_Error	 := TRUE;
	_ErrorId := _McMoveAbs.ErrorID;
END_IF

_McMoveAbs.Execute := FALSE;

